LIN {X 0,Y 419.556,Z 514.347,A -85,B 0,C 180,E1 -10185.297,E2 -10185.297} C_VEL
LIN {X 0,Y 420.532,Z 504.922,A -85,B 0,C 180,E1 -10186.755,E2 -10186.755} C_VEL
LIN {X 0,Y 421.766,Z 492.891,A -85,B 0,C 180,E1 -10188.309,E2 -10188.309} C_VEL
LIN {X 0,Y 423.026,Z 480.248,A -85,B 0,C 180,E1 -10189.659,E2 -10189.659} C_VEL
LIN {X 0,Y 424.183,Z 467.994,A -85,B 0,C 180,E1 -10190.741,E2 -10190.741} C_VEL
LIN {X 0,Y 425.391,Z 454.765,A -85,B 0,C 180,E1 -10191.694,E2 -10191.694} C_VEL
LIN {X 0,Y 426.558,Z 439.892,A -85,B 0,C 180,E1 -10192.546,E2 -10192.546} C_VEL
LIN {X 0,Y 427.411,Z 424.917,A -85,B 0,C 180,E1 -10193.196,E2 -10193.196} C_VEL
LIN {X 0,Y 428.173,Z 409.767,A -85,B 0,C 180,E1 -10193.647,E2 -10193.647} C_VEL
LIN {X 0,Y 428.857,Z 376.254,A -85,B 0,C 180,E1 -10194.249,E2 -10194.249} C_VEL
LIN {X 0,Y 430.577,Z 275.254,A -85,B 0,C 180,E1 -10195.966,E2 -10195.966} C_VEL
LIN {X 0,Y 425.192,Z 246.932,A -85,B 0,C 180,E1 -10196.839,E2 -10196.839} C_VEL
LIN {X 0,Y 424.129,Z 241.646,A -85,B 0,C 180,E1 -10197.03,E2 -10197.03} C_VEL
LIN {X 0,Y 424.477,Z 235.443,A -85,B 0,C 180,E1 -10198.074,E2 -10198.074} C_VEL
LIN {X 0,Y 421.44,Z 222.358,A -85,B 0,C 180,E1 -10200.571,E2 -10200.571} C_VEL
LIN {X 0,Y 418.245,Z 209.999,A -85,B 0,C 180,E1 -10203.07,E2 -10203.07} C_VEL
LIN {X 0,Y 418.245,Z 210.011,A -85,B 0,C 180,E1 -10206.238,E2 -10206.238} C_VEL
LIN {X 0,Y 418.26,Z 210.01,A -85,B 0,C 180,E1 -10209.68,E2 -10209.68} C_VEL
LIN {X 0,Y 418.241,Z 210.012,A -85,B 0,C 180,E1 -10212.323,E2 -10212.323} C_VEL
LIN {X 0,Y 418.23,Z 210.009,A -85,B 0,C 180,E1 -10215.108,E2 -10215.108} C_VEL
LIN {X 0,Y 418.251,Z 210.009,A -85,B 0,C 180,E1 -10217.768,E2 -10217.768} C_VEL
LIN {X 0,Y 418.261,Z 210.005,A -85,B 0,C 180,E1 -10220.616,E2 -10220.616} C_VEL
LIN {X 0,Y 418.24,Z 210.008,A -85,B 0,C 180,E1 -10223.976,E2 -10223.976} C_VEL
LIN {X 0,Y 418.253,Z 210.004,A -85,B 0,C 180,E1 -10227.155,E2 -10227.155} C_VEL
LIN {X 0,Y 418.267,Z 210.003,A -85,B 0,C 180,E1 -10230.838,E2 -10230.838} C_VEL
LIN {X 0,Y 418.263,Z 210.01,A -85,B 0,C 180,E1 -10234.096,E2 -10234.096} C_VEL
LIN {X 0,Y 418.224,Z 210.004,A -85,B 0,C 180,E1 -10237.263,E2 -10237.263} C_VEL
LIN {X 0,Y 418.275,Z 210.003,A -85,B 0,C 180,E1 -10240.364,E2 -10240.364} C_VEL
LIN {X 0,Y 418.308,Z 210.002,A -85,B 0,C 180,E1 -10243.404,E2 -10243.404} C_VEL
LIN {X 0,Y 418.338,Z 209.997,A -85,B 0,C 180,E1 -10246.999,E2 -10246.999} C_VEL
LIN {X 0,Y 418.334,Z 209.997,A -85,B 0,C 180,E1 -10250.329,E2 -10250.329} C_VEL
LIN {X 0,Y 418.484,Z 209.981,A -85,B 0,C 180,E1 -10253.249,E2 -10253.249} C_VEL
LIN {X 0,Y 418.333,Z 210,A -85,B 0,C 180,E1 -10255.182,E2 -10255.182} C_VEL
LIN {X 0,Y 418.536,Z 209.973,A -85,B 0,C 180,E1 -10258.076,E2 -10258.076} C_VEL
LIN {X 0,Y 418.665,Z 209.953,A -85,B 0,C 180,E1 -10260,E2 -10260} C_VEL
LIN {X 0,Y 418.503,Z 209.979,A -85,B 0,C 180,E1 -10262.888,E2 -10262.888} C_VEL
LIN {X 0,Y 418.486,Z 209.98,A -85,B 0,C 180,E1 -10266.751,E2 -10266.751} C_VEL
LIN {X 0,Y 418.334,Z 210,A -85,B 0,C 180,E1 -10269.672,E2 -10269.672} C_VEL
LIN {X 0,Y 418.339,Z 209.996,A -85,B 0,C 180,E1 -10273.001,E2 -10273.001} C_VEL
LIN {X 0,Y 418.305,Z 210.001,A -85,B 0,C 180,E1 -10276.736,E2 -10276.736} C_VEL
LIN {X 0,Y 418.263,Z 210.005,A -85,B 0,C 180,E1 -10279.791,E2 -10279.791} C_VEL
LIN {X 0,Y 418.225,Z 210.014,A -85,B 0,C 180,E1 -10282.737,E2 -10282.737} C_VEL
LIN {X 0,Y 418.263,Z 209.987,A -85,B 0,C 180,E1 -10285.905,E2 -10285.905} C_VEL
LIN {X 0,Y 418.269,Z 210.011,A -85,B 0,C 180,E1 -10289.162,E2 -10289.162} C_VEL
LIN {X 0,Y 418.252,Z 210.013,A -85,B 0,C 180,E1 -10292.845,E2 -10292.845} C_VEL
LIN {X 0,Y 418.243,Z 210.009,A -85,B 0,C 180,E1 -10296.239,E2 -10296.239} C_VEL
LIN {X 0,Y 418.244,Z 210.006,A -85,B 0,C 180,E1 -10299.683,E2 -10299.683} C_VEL
LIN {X 0,Y 418.227,Z 210.009,A -85,B 0,C 180,E1 -10302.322,E2 -10302.322} C_VEL
LIN {X 0,Y 418.238,Z 210.013,A -85,B 0,C 180,E1 -10305.11,E2 -10305.11} C_VEL
LIN {X 0,Y 418.239,Z 210.011,A -85,B 0,C 180,E1 -10307.768,E2 -10307.768} C_VEL
LIN {X 0,Y 418.255,Z 210.007,A -85,B 0,C 180,E1 -10310.619,E2 -10310.619} C_VEL
LIN {X 0,Y 418.24,Z 210.008,A -85,B 0,C 180,E1 -10313.977,E2 -10313.977} C_VEL
LIN {X 0,Y 418.256,Z 210.009,A -85,B 0,C 180,E1 -10317.157,E2 -10317.157} C_VEL
LIN {X 0,Y 418.269,Z 210.134,A -85,B 0,C 180,E1 -10320.425,E2 -10320.425} C_VEL
LIN {X 0,Y 421.107,Z 221.313,A -85,B 0,C 180,E1 -10322.844,E2 -10322.844} C_VEL
LIN {X 0,Y 429.206,Z 240.547,A -85,B 0,C 180,E1 -10323.755,E2 -10323.755} C_VEL
LIN {X 0,Y 430.885,Z 248.586,A -85,B 0,C 180,E1 -10324.013,E2 -10324.013} C_VEL
LIN {X 0,Y 429.161,Z 353.4,A -85,B 0,C 180,E1 -10325.801,E2 -10325.801} C_VEL
LIN {X 0,Y 428.505,Z 387.1,A -85,B 0,C 180,E1 -10326.404,E2 -10326.404} C_VEL
LIN {X 0,Y 427.927,Z 402.384,A -85,B 0,C 180,E1 -10326.867,E2 -10326.867} C_VEL
LIN {X 0,Y 427.22,Z 415.712,A -85,B 0,C 180,E1 -10327.435,E2 -10327.435} C_VEL
LIN {X 0,Y 426.193,Z 429.869,A -85,B 0,C 180,E1 -10328.221,E2 -10328.221} C_VEL
LIN {X 0,Y 425.1,Z 443.449,A -85,B 0,C 180,E1 -10329.179,E2 -10329.179} C_VEL
LIN {X 0,Y 423.774,Z 457.224,A -85,B 0,C 180,E1 -10330.377,E2 -10330.377} C_VEL
LIN {X 0,Y 422.655,Z 468.581,A -85,B 0,C 180,E1 -10331.583,E2 -10331.583} C_VEL
LIN {X 0,Y 421.421,Z 480.043,A -85,B 0,C 180,E1 -10333.032,E2 -10333.032} C_VEL
LIN {X 0,Y 421.245,Z 481.801,A -85,B 0,C 180,E1 -10333.273,E2 -10333.273} C_VEL
LIN {X 0,Y 420.192,Z 485.905,A -85,B 0,C 180,E1 -10333.835,E2 -10333.835} C_VEL
LIN {X 0,Y 416.726,Z 492.332,A -85,B 0,C 180,E1 -10334.755,E2 -10334.755} C_VEL
LIN {X 0,Y 413.246,Z 498.267,A -85,B 0,C 180,E1 -10335.744,E2 -10335.744} C_VEL
LIN {X 0,Y 412.186,Z 501.6,A -85,B 0,C 180,E1 -10336.407,E2 -10336.407} C_VEL
LIN {X 0,Y 411.566,Z 509.194,A -85,B 0,C 180,E1 -10338.176,E2 -10338.176} C_VEL
LIN {X 0,Y 410.838,Z 516.135,A -85,B 0,C 180,E1 -10340.15,E2 -10340.15} C_VEL
LIN {X 0,Y 410.44,Z 521.585,A -85,B 0,C 180,E1 -10342.127,E2 -10342.127} C_VEL
LIN {X 0,Y 410.201,Z 525.699,A -85,B 0,C 180,E1 -10344.1,E2 -10344.1} C_VEL
LIN {X 0,Y 409.982,Z 528.593,A -85,B 0,C 180,E1 -10346.068,E2 -10346.068} C_VEL
LIN {X 0,Y 410.007,Z 530.331,A -85,B 0,C 180,E1 -10348.035,E2 -10348.035} C_VEL
LIN {X 0,Y 409.925,Z 530.941,A -85,B 0,C 180,E1 -10350,E2 -10350} C_VEL
LIN {X 0,Y 410.008,Z 530.379,A -85,B 0,C 180,E1 -10351.965,E2 -10351.965} C_VEL
LIN {X 0,Y 409.981,Z 528.706,A -85,B 0,C 180,E1 -10353.932,E2 -10353.932} C_VEL
LIN {X 0,Y 410.185,Z 525.873,A -85,B 0,C 180,E1 -10355.9,E2 -10355.9} C_VEL
LIN {X 0,Y 410.411,Z 521.819,A -85,B 0,C 180,E1 -10357.874,E2 -10357.874} C_VEL
LIN {X 0,Y 410.824,Z 516.442,A -85,B 0,C 180,E1 -10359.85,E2 -10359.85} C_VEL
LIN {X 0,Y 411.55,Z 509.585,A -85,B 0,C 180,E1 -10361.825,E2 -10361.825} C_VEL
LIN {X 0,Y 412.292,Z 501.03,A -85,B 0,C 180,E1 -10363.806,E2 -10363.806} C_VEL
LIN {X 0,Y 413.317,Z 491.928,A -85,B 0,C 180,E1 -10365.534,E2 -10365.534} C_VEL
LIN {X 0,Y 414.339,Z 482.65,A -85,B 0,C 180,E1 -10367.013,E2 -10367.013} C_VEL
LIN {X 0,Y 415.663,Z 470.729,A -85,B 0,C 180,E1 -10368.6,E2 -10368.6} C_VEL
LIN {X 0,Y 417.002,Z 458.382,A -85,B 0,C 180,E1 -10369.955,E2 -10369.955} C_VEL
LIN {X 0,Y 418.359,Z 444.849,A -85,B 0,C 180,E1 -10371.172,E2 -10371.172} C_VEL
LIN {X 0,Y 419.529,Z 431.537,A -85,B 0,C 180,E1 -10372.143,E2 -10372.143} C_VEL
LIN {X 0,Y 420.595,Z 416.874,A -85,B 0,C 180,E1 -10372.988,E2 -10372.988} C_VEL
LIN {X 0,Y 421.415,Z 402.214,A -85,B 0,C 180,E1 -10373.626,E2 -10373.626} C_VEL
LIN {X 0,Y 422.043,Z 387.314,A -85,B 0,C 180,E1 -10374.077,E2 -10374.077} C_VEL
LIN {X 0,Y 422.876,Z 348.258,A -85,B 0,C 180,E1 -10374.779,E2 -10374.779} C_VEL
LIN {X 0,Y 424.496,Z 248.846,A -85,B 0,C 180,E1 -10376.506,E2 -10376.506} C_VEL
LIN {X 0,Y 422.718,Z 241.83,A -85,B 0,C 180,E1 -10376.758,E2 -10376.758} C_VEL
LIN {X 0,Y 414.382,Z 222.693,A -85,B 0,C 180,E1 -10377.712,E2 -10377.712} C_VEL
LIN {X 0,Y 413.816,Z 221.203,A -85,B 0,C 180,E1 -10377.806,E2 -10377.806} C_VEL
LIN {X 0,Y 411.215,Z 210.89,A -85,B 0,C 180,E1 -10380.134,E2 -10380.134} C_VEL
LIN {X 0,Y 411.205,Z 210.895,A -85,B 0,C 180,E1 -10383.155,E2 -10383.155} C_VEL
LIN {X 0,Y 411.193,Z 210.888,A -85,B 0,C 180,E1 -10386.552,E2 -10386.552} C_VEL
LIN {X 0,Y 411.211,Z 210.883,A -85,B 0,C 180,E1 -10389.727,E2 -10389.727} C_VEL
LIN {X 0,Y 411.174,Z 210.894,A -85,B 0,C 180,E1 -10393.132,E2 -10393.132} C_VEL
LIN {X 0,Y 411.164,Z 210.891,A -85,B 0,C 180,E1 -10395.88,E2 -10395.88} C_VEL
LIN {X 0,Y 411.195,Z 210.883,A -85,B 0,C 180,E1 -10398.765,E2 -10398.765} C_VEL
LIN {X 0,Y 411.198,Z 210.876,A -85,B 0,C 180,E1 -10402.027,E2 -10402.027} C_VEL
LIN {X 0,Y 411.2,Z 210.888,A -85,B 0,C 180,E1 -10405.666,E2 -10405.666} C_VEL
LIN {X 0,Y 411.191,Z 210.874,A -85,B 0,C 180,E1 -10409.152,E2 -10409.152} C_VEL
LIN {X 0,Y 411.253,Z 210.882,A -85,B 0,C 180,E1 -10412.522,E2 -10412.522} C_VEL
LIN {X 0,Y 411.219,Z 210.884,A -85,B 0,C 180,E1 -10415.784,E2 -10415.784} C_VEL
LIN {X 0,Y 411.188,Z 210.892,A -85,B 0,C 180,E1 -10418.965,E2 -10418.965} C_VEL
LIN {X 0,Y 411.245,Z 210.877,A -85,B 0,C 180,E1 -10422.084,E2 -10422.084} C_VEL
LIN {X 0,Y 411.252,Z 210.877,A -85,B 0,C 180,E1 -10425.147,E2 -10425.147} C_VEL
LIN {X 0,Y 411.277,Z 210.878,A -85,B 0,C 180,E1 -10428.167,E2 -10428.167} C_VEL
LIN {X 0,Y 411.432,Z 210.858,A -85,B 0,C 180,E1 -10432.189,E2 -10432.189} C_VEL
LIN {X 0,Y 411.466,Z 210.852,A -85,B 0,C 180,E1 -10434.118,E2 -10434.118} C_VEL
LIN {X 0,Y 411.505,Z 210.849,A -85,B 0,C 180,E1 -10438.042,E2 -10438.042} C_VEL
LIN {X 0,Y 411.635,Z 210.827,A -85,B 0,C 180,E1 -10440,E2 -10440} C_VEL
LIN {X 0,Y 411.458,Z 210.853,A -85,B 0,C 180,E1 -10442.937,E2 -10442.937} C_VEL
LIN {X 0,Y 411.447,Z 210.857,A -85,B 0,C 180,E1 -10446.867,E2 -10446.867} C_VEL
LIN {X 0,Y 411.285,Z 210.875,A -85,B 0,C 180,E1 -10449.839,E2 -10449.839} C_VEL
LIN {X 0,Y 411.297,Z 210.872,A -85,B 0,C 180,E1 -10453.104,E2 -10453.104} C_VEL
LIN {X 0,Y 411.255,Z 210.883,A -85,B 0,C 180,E1 -10455.868,E2 -10455.868} C_VEL
LIN {X 0,Y 411.217,Z 210.888,A -85,B 0,C 180,E1 -10458.949,E2 -10458.949} C_VEL
LIN {X 0,Y 411.196,Z 210.892,A -85,B 0,C 180,E1 -10462.643,E2 -10462.643} C_VEL
LIN {X 0,Y 411.229,Z 210.88,A -85,B 0,C 180,E1 -10465.293,E2 -10465.293} C_VEL
LIN {X 0,Y 411.217,Z 210.889,A -85,B 0,C 180,E1 -10468.59,E2 -10468.59} C_VEL
LIN {X 0,Y 411.164,Z 210.894,A -85,B 0,C 180,E1 -10471.997,E2 -10471.997} C_VEL
LIN {X 0,Y 411.192,Z 210.888,A -85,B 0,C 180,E1 -10475.529,E2 -10475.529} C_VEL
LIN {X 0,Y 411.212,Z 210.881,A -85,B 0,C 180,E1 -10479.225,E2 -10479.225} C_VEL
LIN {X 0,Y 411.176,Z 210.892,A -85,B 0,C 180,E1 -10482.696,E2 -10482.696} C_VEL
LIN {X 0,Y 411.163,Z 210.895,A -85,B 0,C 180,E1 -10485.882,E2 -10485.882} C_VEL
LIN {X 0,Y 411.196,Z 210.888,A -85,B 0,C 180,E1 -10488.766,E2 -10488.766} C_VEL
LIN {X 0,Y 411.2,Z 210.882,A -85,B 0,C 180,E1 -10492.028,E2 -10492.028} C_VEL
LIN {X 0,Y 411.203,Z 210.89,A -85,B 0,C 180,E1 -10495.667,E2 -10495.667} C_VEL
LIN {X 0,Y 411.209,Z 210.944,A -85,B 0,C 180,E1 -10496.516,E2 -10496.516} C_VEL
LIN {X 0,Y 415.204,Z 226.483,A -85,B 0,C 180,E1 -10499.684,E2 -10499.684} C_VEL
LIN {X 0,Y 417.712,Z 237.94,A -85,B 0,C 180,E1 -10501.895,E2 -10501.895} C_VEL
LIN {X 0,Y 417.473,Z 241.807,A -85,B 0,C 180,E1 -10502.522,E2 -10502.522} C_VEL
LIN {X 0,Y 423.749,Z 273.294,A -85,B 0,C 180,E1 -10503.543,E2 -10503.543} C_VEL
LIN {X 0,Y 424.228,Z 277.071,A -85,B 0,C 180,E1 -10503.645,E2 -10503.645} C_VEL
LIN {X 0,Y 421.757,Z 407.384,A -85,B 0,C 180,E1 -10505.905,E2 -10505.905} C_VEL
LIN {X 0,Y 421.078,Z 422.903,A -85,B 0,C 180,E1 -10506.354,E2 -10506.354} C_VEL
LIN {X 0,Y 420.16,Z 437.166,A -85,B 0,C 180,E1 -10506.95,E2 -10506.95} C_VEL
LIN {X 0,Y 419.122,Z 450.867,A -85,B 0,C 180,E1 -10507.705,E2 -10507.705} C_VEL
LIN {X 0,Y 417.804,Z 464.768,A -85,B 0,C 180,E1 -10508.669,E2 -10508.669} C_VEL
LIN {X 0,Y 416.602,Z 477.512,A -85,B 0,C 180,E1 -10509.768,E2 -10509.768} C_VEL
LIN {X 0,Y 415.151,Z 490.399,A -85,B 0,C 180,E1 -10511.11,E2 -10511.11} C_VEL
LIN {X 0,Y 414.054,Z 501.198,A -85,B 0,C 180,E1 -10512.466,E2 -10512.466} C_VEL
LIN {X 0,Y 412.908,Z 511.188,A -85,B 0,C 180,E1 -10513.944,E2 -10513.944} C_VEL
LIN {X 0,Y 411.914,Z 520.968,A -85,B 0,C 180,E1 -10515.677,E2 -10515.677} C_VEL
LIN {X 0,Y 411.211,Z 529.133,A -85,B 0,C 180,E1 -10517.414,E2 -10517.414} C_VEL
LIN {X 0,Y 410.667,Z 535.884,A -85,B 0,C 180,E1 -10519.15,E2 -10519.15} C_VEL
LIN {X 0,Y 410.235,Z 542.121,A -85,B 0,C 180,E1 -10521.131,E2 -10521.131} C_VEL
LIN {X 0,Y 410.056,Z 546.949,A -85,B 0,C 180,E1 -10523.11,E2 -10523.11} C_VEL
LIN {X 0,Y 409.935,Z 550.485,A -85,B 0,C 180,E1 -10525.083,E2 -10525.083} C_VEL
LIN {X 0,Y 409.903,Z 552.813,A -85,B 0,C 180,E1 -10527.052,E2 -10527.052} C_VEL
LIN {X 0,Y 409.933,Z 553.984,A -85,B 0,C 180,E1 -10529.018,E2 -10529.018} C_VEL
LIN {X 0,Y 409.933,Z 553.983,A -85,B 0,C 180,E1 -10530.982,E2 -10530.982} C_VEL
LIN {X 0,Y 409.903,Z 552.804,A -85,B 0,C 180,E1 -10532.948,E2 -10532.948} C_VEL
LIN {X 0,Y 409.939,Z 550.474,A -85,B 0,C 180,E1 -10534.917,E2 -10534.917} C_VEL
LIN {X 0,Y 410.06,Z 546.939,A -85,B 0,C 180,E1 -10536.89,E2 -10536.89} C_VEL
LIN {X 0,Y 410.235,Z 542.11,A -85,B 0,C 180,E1 -10538.869,E2 -10538.869} C_VEL
LIN {X 0,Y 410.667,Z 535.86,A -85,B 0,C 180,E1 -10540.85,E2 -10540.85} C_VEL
LIN {X 0,Y 411.177,Z 529.103,A -85,B 0,C 180,E1 -10542.587,E2 -10542.587} C_VEL
LIN {X 0,Y 411.912,Z 520.937,A -85,B 0,C 180,E1 -10544.323,E2 -10544.323} C_VEL
LIN {X 0,Y 412.912,Z 511.152,A -85,B 0,C 180,E1 -10546.056,E2 -10546.056} C_VEL
LIN {X 0,Y 414.048,Z 501.152,A -85,B 0,C 180,E1 -10547.534,E2 -10547.534} C_VEL
LIN {X 0,Y 415.294,Z 489.277,A -85,B 0,C 180,E1 -10549.012,E2 -10549.012} C_VEL
LIN {X 0,Y 416.592,Z 477.449,A -85,B 0,C 180,E1 -10550.233,E2 -10550.233} C_VEL
LIN {X 0,Y 417.846,Z 464.677,A -85,B 0,C 180,E1 -10551.329,E2 -10551.329} C_VEL
LIN {X 0,Y 419.092,Z 450.747,A -85,B 0,C 180,E1 -10552.297,E2 -10552.297} C_VEL
LIN {X 0,Y 420.238,Z 435.912,A -85,B 0,C 180,E1 -10553.102,E2 -10553.102} C_VEL
LIN {X 0,Y 421.135,Z 420.871,A -85,B 0,C 180,E1 -10553.708,E2 -10553.708} C_VEL
LIN {X 0,Y 421.828,Z 405.525,A -85,B 0,C 180,E1 -10554.123,E2 -10554.123} C_VEL
LIN {X 0,Y 424.192,Z 276.094,A -85,B 0,C 180,E1 -10556.367,E2 -10556.367} C_VEL
LIN {X 0,Y 418.811,Z 248.109,A -85,B 0,C 180,E1 -10557.255,E2 -10557.255} C_VEL
LIN {X 0,Y 417.458,Z 241.434,A -85,B 0,C 180,E1 -10557.499,E2 -10557.499} C_VEL
LIN {X 0,Y 417.705,Z 237.876,A -85,B 0,C 180,E1 -10558.106,E2 -10558.106} C_VEL
LIN {X 0,Y 415.22,Z 226.384,A -85,B 0,C 180,E1 -10560.32,E2 -10560.32} C_VEL
LIN {X 0,Y 411.212,Z 210.874,A -85,B 0,C 180,E1 -10563.52,E2 -10563.52} C_VEL
LIN {X 0,Y 411.19,Z 210.89,A -85,B 0,C 180,E1 -10566.741,E2 -10566.741} C_VEL
LIN {X 0,Y 411.223,Z 210.886,A -85,B 0,C 180,E1 -10569.729,E2 -10569.729} C_VEL
LIN {X 0,Y 411.173,Z 210.889,A -85,B 0,C 180,E1 -10573.132,E2 -10573.132} C_VEL
LIN {X 0,Y 411.163,Z 210.894,A -85,B 0,C 180,E1 -10575.88,E2 -10575.88} C_VEL
LIN {X 0,Y 411.194,Z 210.885,A -85,B 0,C 180,E1 -10578.765,E2 -10578.765} C_VEL
LIN {X 0,Y 411.198,Z 210.886,A -85,B 0,C 180,E1 -10582.027,E2 -10582.027} C_VEL
LIN {X 0,Y 411.2,Z 210.887,A -85,B 0,C 180,E1 -10585.666,E2 -10585.666} C_VEL
LIN {X 0,Y 411.193,Z 210.886,A -85,B 0,C 180,E1 -10589.153,E2 -10589.153} C_VEL
LIN {X 0,Y 411.253,Z 210.877,A -85,B 0,C 180,E1 -10592.522,E2 -10592.522} C_VEL
LIN {X 0,Y 411.213,Z 210.886,A -85,B 0,C 180,E1 -10595.784,E2 -10595.784} C_VEL
LIN {X 0,Y 411.188,Z 210.872,A -85,B 0,C 180,E1 -10598.966,E2 -10598.966} C_VEL
LIN {X 0,Y 411.244,Z 210.882,A -85,B 0,C 180,E1 -10602.085,E2 -10602.085} C_VEL
LIN {X 0,Y 411.251,Z 210.881,A -85,B 0,C 180,E1 -10605.147,E2 -10605.147} C_VEL
LIN {X 0,Y 411.276,Z 210.876,A -85,B 0,C 180,E1 -10608.167,E2 -10608.167} C_VEL
LIN {X 0,Y 411.432,Z 210.856,A -85,B 0,C 180,E1 -10612.189,E2 -10612.189} C_VEL
LIN {X 0,Y 411.466,Z 210.853,A -85,B 0,C 180,E1 -10614.118,E2 -10614.118} C_VEL
LIN {X 0,Y 411.505,Z 210.849,A -85,B 0,C 180,E1 -10618.043,E2 -10618.043} C_VEL
LIN {X 0,Y 411.635,Z 210.828,A -85,B 0,C 180,E1 -10620,E2 -10620} C_VEL
LIN {X 0,Y 411.458,Z 210.857,A -85,B 0,C 180,E1 -10622.937,E2 -10622.937} C_VEL
LIN {X 0,Y 411.453,Z 210.857,A -85,B 0,C 180,E1 -10626.867,E2 -10626.867} C_VEL
LIN {X 0,Y 411.286,Z 210.877,A -85,B 0,C 180,E1 -10629.839,E2 -10629.839} C_VEL
LIN {X 0,Y 411.298,Z 210.873,A -85,B 0,C 180,E1 -10633.105,E2 -10633.105} C_VEL
LIN {X 0,Y 411.255,Z 210.879,A -85,B 0,C 180,E1 -10636.869,E2 -10636.869} C_VEL
LIN {X 0,Y 411.223,Z 210.881,A -85,B 0,C 180,E1 -10639.987,E2 -10639.987} C_VEL
LIN {X 0,Y 411.189,Z 210.891,A -85,B 0,C 180,E1 -10643.148,E2 -10643.148} C_VEL
LIN {X 0,Y 411.231,Z 210.863,A -85,B 0,C 180,E1 -10646.381,E2 -10646.381} C_VEL
LIN {X 0,Y 411.205,Z 210.886,A -85,B 0,C 180,E1 -10649.712,E2 -10649.712} C_VEL
LIN {X 0,Y 411.201,Z 210.887,A -85,B 0,C 180,E1 -10653.156,E2 -10653.156} C_VEL
LIN {X 0,Y 411.19,Z 210.889,A -85,B 0,C 180,E1 -10656.554,E2 -10656.554} C_VEL
LIN {X 0,Y 411.208,Z 210.882,A -85,B 0,C 180,E1 -10659.729,E2 -10659.729} C_VEL
LIN {X 0,Y 411.173,Z 210.891,A -85,B 0,C 180,E1 -10663.134,E2 -10663.134} C_VEL
LIN {X 0,Y 411.17,Z 210.89,A -85,B 0,C 180,E1 -10665.881,E2 -10665.881} C_VEL
LIN {X 0,Y 411.163,Z 210.896,A -85,B 0,C 180,E1 -10668.772,E2 -10668.772} C_VEL
LIN {X 0,Y 411.204,Z 210.886,A -85,B 0,C 180,E1 -10671.832,E2 -10671.832} C_VEL
LIN {X 0,Y 411.208,Z 210.891,A -85,B 0,C 180,E1 -10675.122,E2 -10675.122} C_VEL
LIN {X 0,Y 411.164,Z 210.896,A -85,B 0,C 180,E1 -10678.003,E2 -10678.003} C_VEL
LIN {X 0,Y 411.239,Z 211.022,A -85,B 0,C 180,E1 -10680.009,E2 -10680.009} C_VEL
LIN {X 0,Y 413.982,Z 221.604,A -85,B 0,C 180,E1 -10682.338,E2 -10682.338} C_VEL
LIN {X 0,Y 423.128,Z 243.066,A -85,B 0,C 180,E1 -10683.392,E2 -10683.392} C_VEL
LIN {X 0,Y 424.523,Z 249.367,A -85,B 0,C 180,E1 -10683.604,E2 -10683.604} C_VEL
LIN {X 0,Y 422.698,Z 353.627,A -85,B 0,C 180,E1 -10685.407,E2 -10685.407} C_VEL
LIN {X 0,Y 422.011,Z 387.317,A -85,B 0,C 180,E1 -10686.018,E2 -10686.018} C_VEL
LIN {X 0,Y 421.407,Z 402.714,A -85,B 0,C 180,E1 -10686.492,E2 -10686.492} C_VEL
LIN {X 0,Y 420.653,Z 416.329,A -85,B 0,C 180,E1 -10687.083,E2 -10687.083} C_VEL
LIN {X 0,Y 419.607,Z 430.077,A -85,B 0,C 180,E1 -10687.862,E2 -10687.862} C_VEL
LIN {X 0,Y 418.479,Z 443.656,A -85,B 0,C 180,E1 -10688.834,E2 -10688.834} C_VEL
LIN {X 0,Y 417.067,Z 457.431,A -85,B 0,C 180,E1 -10690.048,E2 -10690.048} C_VEL
LIN {X 0,Y 415.783,Z 469.85,A -85,B 0,C 180,E1 -10691.395,E2 -10691.395} C_VEL
LIN {X 0,Y 414.618,Z 480.247,A -85,B 0,C 180,E1 -10692.745,E2 -10692.745} C_VEL
LIN {X 0,Y 413.534,Z 489.888,A -85,B 0,C 180,E1 -10694.222,E2 -10694.222} C_VEL
LIN {X 0,Y 412.463,Z 499.336,A -85,B 0,C 180,E1 -10695.948,E2 -10695.948} C_VEL
LIN {X 0,Y 412.186,Z 501.6,A -85,B 0,C 180,E1 -10696.407,E2 -10696.407} C_VEL
LIN {X 0,Y 411.167,Z 504.821,A -85,B 0,C 180,E1 -10697.086,E2 -10697.086} C_VEL
LIN {X 0,Y 407.865,Z 509.804,A -85,B 0,C 180,E1 -10698.194,E2 -10698.194} C_VEL
LIN {X 0,Y 404.646,Z 514.3,A -85,B 0,C 180,E1 -10699.354,E2 -10699.354} C_VEL
LIN {X 0,Y 403.77,Z 516.725,A -85,B 0,C 180,E1 -10700.108,E2 -10700.108} C_VEL
LIN {X 0,Y 403.388,Z 521.787,A -85,B 0,C 180,E1 -10701.988,E2 -10701.988} C_VEL
LIN {X 0,Y 403.122,Z 525.901,A -85,B 0,C 180,E1 -10703.996,E2 -10703.996} C_VEL
LIN {X 0,Y 402.902,Z 528.794,A -85,B 0,C 180,E1 -10705.999,E2 -10705.999} C_VEL
LIN {X 0,Y 402.921,Z 530.531,A -85,B 0,C 180,E1 -10708.001,E2 -10708.001} C_VEL
LIN {X 0,Y 402.85,Z 531.141,A -85,B 0,C 180,E1 -10710,E2 -10710} C_VEL
LIN {X 0,Y 402.921,Z 530.579,A -85,B 0,C 180,E1 -10711.999,E2 -10711.999} C_VEL
LIN {X 0,Y 402.901,Z 528.906,A -85,B 0,C 180,E1 -10714.001,E2 -10714.001} C_VEL
LIN {X 0,Y 403.109,Z 526.073,A -85,B 0,C 180,E1 -10716.004,E2 -10716.004} C_VEL
LIN {X 0,Y 403.366,Z 522.019,A -85,B 0,C 180,E1 -10718.012,E2 -10718.012} C_VEL
LIN {X 0,Y 403.794,Z 516.643,A -85,B 0,C 180,E1 -10720.023,E2 -10720.023} C_VEL
LIN {X 0,Y 404.586,Z 509.785,A -85,B 0,C 180,E1 -10722.031,E2 -10722.031} C_VEL
LIN {X 0,Y 405.386,Z 501.229,A -85,B 0,C 180,E1 -10724.046,E2 -10724.046} C_VEL
LIN {X 0,Y 406.436,Z 492.127,A -85,B 0,C 180,E1 -10725.803,E2 -10725.803} C_VEL
LIN {X 0,Y 407.518,Z 482.849,A -85,B 0,C 180,E1 -10727.307,E2 -10727.307} C_VEL
LIN {X 0,Y 408.843,Z 471.501,A -85,B 0,C 180,E1 -10728.846,E2 -10728.846} C_VEL
LIN {X 0,Y 410.335,Z 458.579,A -85,B 0,C 180,E1 -10730.293,E2 -10730.293} C_VEL
LIN {X 0,Y 411.716,Z 445.045,A -85,B 0,C 180,E1 -10731.53,E2 -10731.53} C_VEL
LIN {X 0,Y 412.968,Z 431.731,A -85,B 0,C 180,E1 -10732.514,E2 -10732.514} C_VEL
LIN {X 0,Y 414.105,Z 416.59,A -85,B 0,C 180,E1 -10733.396,E2 -10733.396} C_VEL
LIN {X 0,Y 414.969,Z 401.595,A -85,B 0,C 180,E1 -10734.049,E2 -10734.049} C_VEL
LIN {X 0,Y 415.631,Z 386.311,A -85,B 0,C 180,E1 -10734.506,E2 -10734.506} C_VEL
LIN {X 0,Y 417.65,Z 282.682,A -85,B 0,C 180,E1 -10736.341,E2 -10736.341} C_VEL
LIN {X 0,Y 418.218,Z 250.264,A -85,B 0,C 180,E1 -10736.913,E2 -10736.913} C_VEL
LIN {X 0,Y 416.588,Z 244.136,A -85,B 0,C 180,E1 -10737.144,E2 -10737.144} C_VEL
LIN {X 0,Y 407.787,Z 224.161,A -85,B 0,C 180,E1 -10738.175,E2 -10738.175} C_VEL
LIN {X 0,Y 406.59,Z 221.401,A -85,B 0,C 180,E1 -10738.349,E2 -10738.349} C_VEL
LIN {X 0,Y 404.156,Z 211.768,A -85,B 0,C 180,E1 -10740.572,E2 -10740.572} C_VEL
LIN {X 0,Y 404.143,Z 211.768,A -85,B 0,C 180,E1 -10743.812,E2 -10743.812} C_VEL
LIN {X 0,Y 404.137,Z 211.767,A -85,B 0,C 180,E1 -10746.875,E2 -10746.875} C_VEL
LIN {X 0,Y 404.144,Z 211.763,A -85,B 0,C 180,E1 -10750.079,E2 -10750.079} C_VEL
LIN {X 0,Y 404.153,Z 211.768,A -85,B 0,C 180,E1 -10753.084,E2 -10753.084} C_VEL
LIN {X 0,Y 404.144,Z 211.766,A -85,B 0,C 180,E1 -10755.925,E2 -10755.925} C_VEL
LIN {X 0,Y 404.147,Z 211.76,A -85,B 0,C 180,E1 -10758.638,E2 -10758.638} C_VEL
LIN {X 0,Y 404.156,Z 211.756,A -85,B 0,C 180,E1 -10761.49,E2 -10761.49} C_VEL
LIN {X 0,Y 404.18,Z 211.763,A -85,B 0,C 180,E1 -10764.983,E2 -10764.983} C_VEL
LIN {X 0,Y 404.139,Z 211.749,A -85,B 0,C 180,E1 -10768.553,E2 -10768.553} C_VEL
LIN {X 0,Y 404.191,Z 211.76,A -85,B 0,C 180,E1 -10772,E2 -10772} C_VEL
LIN {X 0,Y 404.17,Z 211.766,A -85,B 0,C 180,E1 -10775.334,E2 -10775.334} C_VEL
LIN {X 0,Y 404.131,Z 211.766,A -85,B 0,C 180,E1 -10778.58,E2 -10778.58} C_VEL
LIN {X 0,Y 404.202,Z 211.754,A -85,B 0,C 180,E1 -10781.761,E2 -10781.761} C_VEL
LIN {X 0,Y 404.198,Z 211.758,A -85,B 0,C 180,E1 -10784.882,E2 -10784.882} C_VEL
LIN {X 0,Y 404.249,Z 211.753,A -85,B 0,C 180,E1 -10787.958,E2 -10787.958} C_VEL
LIN {X 0,Y 404.397,Z 211.734,A -85,B 0,C 180,E1 -10792.128,E2 -10792.128} C_VEL
LIN {X 0,Y 404.414,Z 211.73,A -85,B 0,C 180,E1 -10794.015,E2 -10794.015} C_VEL
LIN {X 0,Y 404.474,Z 211.725,A -85,B 0,C 180,E1 -10798.008,E2 -10798.008} C_VEL
LIN {X 0,Y 404.604,Z 211.702,A -85,B 0,C 180,E1 -10800,E2 -10800} C_VEL
LIN {X 0,Y 404.415,Z 211.729,A -85,B 0,C 180,E1 -10802.988,E2 -10802.988} C_VEL
LIN {X 0,Y 404.414,Z 211.733,A -85,B 0,C 180,E1 -10805.985,E2 -10805.985} C_VEL
LIN {X 0,Y 404.283,Z 211.748,A -85,B 0,C 180,E1 -10809.001,E2 -10809.001} C_VEL
LIN {X 0,Y 404.248,Z 211.755,A -85,B 0,C 180,E1 -10812.042,E2 -10812.042} C_VEL
LIN {X 0,Y 404.203,Z 211.761,A -85,B 0,C 180,E1 -10815.118,E2 -10815.118} C_VEL
LIN {X 0,Y 404.202,Z 211.758,A -85,B 0,C 180,E1 -10818.238,E2 -10818.238} C_VEL
LIN {X 0,Y 404.13,Z 211.763,A -85,B 0,C 180,E1 -10821.42,E2 -10821.42} C_VEL
LIN {X 0,Y 404.17,Z 211.762,A -85,B 0,C 180,E1 -10824.666,E2 -10824.666} C_VEL
LIN {X 0,Y 404.191,Z 211.765,A -85,B 0,C 180,E1 -10828,E2 -10828} C_VEL
LIN {X 0,Y 404.139,Z 211.768,A -85,B 0,C 180,E1 -10831.56,E2 -10831.56} C_VEL
LIN {X 0,Y 404.178,Z 211.761,A -85,B 0,C 180,E1 -10835.017,E2 -10835.017} C_VEL
LIN {X 0,Y 404.149,Z 211.762,A -85,B 0,C 180,E1 -10838.757,E2 -10838.757} C_VEL
LIN {X 0,Y 404.117,Z 211.76,A -85,B 0,C 180,E1 -10841.6,E2 -10841.6} C_VEL
LIN {X 0,Y 404.14,Z 211.768,A -85,B 0,C 180,E1 -10844.523,E2 -10844.523} C_VEL
LIN {X 0,Y 404.166,Z 211.764,A -85,B 0,C 180,E1 -10847.301,E2 -10847.301} C_VEL
LIN {X 0,Y 404.165,Z 211.764,A -85,B 0,C 180,E1 -10849.956,E2 -10849.956} C_VEL
LIN {X 0,Y 404.137,Z 211.763,A -85,B 0,C 180,E1 -10853.125,E2 -10853.125} C_VEL
LIN {X 0,Y 404.175,Z 211.912,A -85,B 0,C 180,E1 -10856.079,E2 -10856.079} C_VEL
LIN {X 0,Y 408.299,Z 227.76,A -85,B 0,C 180,E1 -10859.389,E2 -10859.389} C_VEL
LIN {X 0,Y 410.858,Z 239.281,A -85,B 0,C 180,E1 -10861.662,E2 -10861.662} C_VEL
LIN {X 0,Y 410.814,Z 241.557,A -85,B 0,C 180,E1 -10862.037,E2 -10862.037} C_VEL
LIN {X 0,Y 416.834,Z 271.28,A -85,B 0,C 180,E1 -10863.035,E2 -10863.035} C_VEL
LIN {X 0,Y 417.868,Z 277.41,A -85,B 0,C 180,E1 -10863.222,E2 -10863.222} C_VEL
LIN {X 0,Y 415.325,Z 405.694,A -85,B 0,C 180,E1 -10865.474,E2 -10865.474} C_VEL
LIN {X 0,Y 414.702,Z 420.881,A -85,B 0,C 180,E1 -10865.901,E2 -10865.901} C_VEL
LIN {X 0,Y 413.81,Z 434.355,A -85,B 0,C 180,E1 -10866.442,E2 -10866.442} C_VEL
LIN {X 0,Y 412.696,Z 448.678,A -85,B 0,C 180,E1 -10867.206,E2 -10867.206} C_VEL
LIN {X 0,Y 411.338,Z 462.985,A -85,B 0,C 180,E1 -10868.185,E2 -10868.185} C_VEL
LIN {X 0,Y 410.039,Z 476.018,A -85,B 0,C 180,E1 -10869.298,E2 -10869.298} C_VEL
LIN {X 0,Y 408.491,Z 489.125,A -85,B 0,C 180,E1 -10870.659,E2 -10870.659} C_VEL
LIN {X 0,Y 407.236,Z 500.997,A -85,B 0,C 180,E1 -10872.162,E2 -10872.162} C_VEL
LIN {X 0,Y 406.009,Z 510.987,A -85,B 0,C 180,E1 -10873.663,E2 -10873.663} C_VEL
LIN {X 0,Y 404.964,Z 520.766,A -85,B 0,C 180,E1 -10875.426,E2 -10875.426} C_VEL
LIN {X 0,Y 404.195,Z 528.931,A -85,B 0,C 180,E1 -10877.192,E2 -10877.192} C_VEL
LIN {X 0,Y 403.655,Z 535.683,A -85,B 0,C 180,E1 -10878.959,E2 -10878.959} C_VEL
LIN {X 0,Y 403.178,Z 541.92,A -85,B 0,C 180,E1 -10880.974,E2 -10880.974} C_VEL
LIN {X 0,Y 402.981,Z 546.748,A -85,B 0,C 180,E1 -10882.988,E2 -10882.988} C_VEL
LIN {X 0,Y 402.851,Z 550.285,A -85,B 0,C 180,E1 -10884.996,E2 -10884.996} C_VEL
LIN {X 0,Y 402.801,Z 552.612,A -85,B 0,C 180,E1 -10887,E2 -10887} C_VEL
LIN {X 0,Y 402.86,Z 553.784,A -85,B 0,C 180,E1 -10889,E2 -10889} C_VEL
LIN {X 0,Y 402.86,Z 553.782,A -85,B 0,C 180,E1 -10891,E2 -10891} C_VEL
LIN {X 0,Y 402.801,Z 552.603,A -85,B 0,C 180,E1 -10893,E2 -10893} C_VEL
LIN {X 0,Y 402.855,Z 550.272,A -85,B 0,C 180,E1 -10895.004,E2 -10895.004} C_VEL
LIN {X 0,Y 402.983,Z 546.737,A -85,B 0,C 180,E1 -10897.012,E2 -10897.012} C_VEL
LIN {X 0,Y 403.178,Z 541.907,A -85,B 0,C 180,E1 -10899.026,E2 -10899.026} C_VEL
LIN {X 0,Y 403.655,Z 535.657,A -85,B 0,C 180,E1 -10901.041,E2 -10901.041} C_VEL
LIN {X 0,Y 404.205,Z 527.807,A -85,B 0,C 180,E1 -10903.063,E2 -10903.063} C_VEL
LIN {X 0,Y 405.122,Z 519.469,A -85,B 0,C 180,E1 -10904.825,E2 -10904.825} C_VEL
LIN {X 0,Y 406.192,Z 509.423,A -85,B 0,C 180,E1 -10906.587,E2 -10906.587} C_VEL
LIN {X 0,Y 407.411,Z 499.155,A -85,B 0,C 180,E1 -10908.089,E2 -10908.089} C_VEL
LIN {X 0,Y 408.808,Z 486.923,A -85,B 0,C 180,E1 -10909.586,E2 -10909.586} C_VEL
LIN {X 0,Y 410.207,Z 474.651,A -85,B 0,C 180,E1 -10910.824,E2 -10910.824} C_VEL
LIN {X 0,Y 411.358,Z 462.883,A -85,B 0,C 180,E1 -10911.814,E2 -10911.814} C_VEL
LIN {X 0,Y 412.696,Z 448.55,A -85,B 0,C 180,E1 -10912.794,E2 -10912.794} C_VEL
LIN {X 0,Y 413.807,Z 434.347,A -85,B 0,C 180,E1 -10913.551,E2 -10913.551} C_VEL
LIN {X 0,Y 414.713,Z 419.744,A -85,B 0,C 180,E1 -10914.131,E2 -10914.131} C_VEL
LIN {X 0,Y 415.372,Z 403.799,A -85,B 0,C 180,E1 -10914.556,E2 -10914.556} C_VEL
LIN {X 0,Y 417.79,Z 278.332,A -85,B 0,C 180,E1 -10916.757,E2 -10916.757} C_VEL
LIN {X 0,Y 417.211,Z 273.692,A -85,B 0,C 180,E1 -10916.884,E2 -10916.884} C_VEL
LIN {X 0,Y 411.403,Z 244.146,A -85,B 0,C 180,E1 -10917.86,E2 -10917.86} C_VEL
LIN {X 0,Y 410.835,Z 241.163,A -85,B 0,C 180,E1 -10917.992,E2 -10917.992} C_VEL
LIN {X 0,Y 410.579,Z 237.65,A -85,B 0,C 180,E1 -10918.638,E2 -10918.638} C_VEL
LIN {X 0,Y 407.577,Z 225.06,A -85,B 0,C 180,E1 -10921.151,E2 -10921.151} C_VEL
LIN {X 0,Y 404.158,Z 211.756,A -85,B 0,C 180,E1 -10923.96,E2 -10923.96} C_VEL
LIN {X 0,Y 404.145,Z 211.769,A -85,B 0,C 180,E1 -10927.49,E2 -10927.49} C_VEL
LIN {X 0,Y 404.162,Z 211.768,A -85,B 0,C 180,E1 -10930.083,E2 -10930.083} C_VEL
LIN {X 0,Y 404.153,Z 211.763,A -85,B 0,C 180,E1 -10933.084,E2 -10933.084} C_VEL
LIN {X 0,Y 404.152,Z 211.762,A -85,B 0,C 180,E1 -10936.915,E2 -10936.915} C_VEL
LIN {X 0,Y 404.163,Z 211.763,A -85,B 0,C 180,E1 -10939.955,E2 -10939.955} C_VEL
LIN {X 0,Y 404.134,Z 211.764,A -85,B 0,C 180,E1 -10943.124,E2 -10943.124} C_VEL
LIN {X 0,Y 404.139,Z 211.764,A -85,B 0,C 180,E1 -10946.187,E2 -10946.187} C_VEL
LIN {X 0,Y 404.148,Z 211.764,A -85,B 0,C 180,E1 -10949.715,E2 -10949.715} C_VEL
LIN {X 0,Y 404.188,Z 211.758,A -85,B 0,C 180,E1 -10953.122,E2 -10953.122} C_VEL
LIN {X 0,Y 404.167,Z 211.765,A -85,B 0,C 180,E1 -10955.334,E2 -10955.334} C_VEL
LIN {X 0,Y 404.13,Z 211.75,A -85,B 0,C 180,E1 -10958.58,E2 -10958.58} C_VEL
LIN {X 0,Y 404.202,Z 211.763,A -85,B 0,C 180,E1 -10961.762,E2 -10961.762} C_VEL
LIN {X 0,Y 404.198,Z 211.758,A -85,B 0,C 180,E1 -10964.882,E2 -10964.882} C_VEL
LIN {X 0,Y 404.249,Z 211.753,A -85,B 0,C 180,E1 -10967.958,E2 -10967.958} C_VEL
LIN {X 0,Y 404.397,Z 211.733,A -85,B 0,C 180,E1 -10972.129,E2 -10972.129} C_VEL
LIN {X 0,Y 404.415,Z 211.732,A -85,B 0,C 180,E1 -10974.015,E2 -10974.015} C_VEL
LIN {X 0,Y 404.474,Z 211.725,A -85,B 0,C 180,E1 -10978.009,E2 -10978.009} C_VEL
LIN {X 0,Y 404.604,Z 211.704,A -85,B 0,C 180,E1 -10980,E2 -10980} C_VEL
LIN {X 0,Y 404.415,Z 211.735,A -85,B 0,C 180,E1 -10982.989,E2 -10982.989} C_VEL
LIN {X 0,Y 404.399,Z 211.737,A -85,B 0,C 180,E1 -10986.988,E2 -10986.988} C_VEL
LIN {X 0,Y 404.251,Z 211.752,A -85,B 0,C 180,E1 -10990.012,E2 -10990.012} C_VEL
LIN {X 0,Y 404.259,Z 211.751,A -85,B 0,C 180,E1 -10993.212,E2 -10993.212} C_VEL
LIN {X 0,Y 404.208,Z 211.757,A -85,B 0,C 180,E1 -10997.007,E2 -10997.007} C_VEL
LIN {X 0,Y 404.156,Z 211.762,A -85,B 0,C 180,E1 -11000.352,E2 -11000.352} C_VEL
LIN {X 0,Y 404.157,Z 211.762,A -85,B 0,C 180,E1 -11003.575,E2 -11003.575} C_VEL
LIN {X 0,Y 404.177,Z 211.741,A -85,B 0,C 180,E1 -11005.767,E2 -11005.767} C_VEL
LIN {X 0,Y 404.192,Z 211.756,A -85,B 0,C 180,E1 -11008,E2 -11008} C_VEL
LIN {X 0,Y 404.137,Z 211.767,A -85,B 0,C 180,E1 -11011.56,E2 -11011.56} C_VEL
LIN {X 0,Y 404.18,Z 211.765,A -85,B 0,C 180,E1 -11015.017,E2 -11015.017} C_VEL
LIN {X 0,Y 404.151,Z 211.766,A -85,B 0,C 180,E1 -11018.757,E2 -11018.757} C_VEL
LIN {X 0,Y 404.119,Z 211.765,A -85,B 0,C 180,E1 -11021.601,E2 -11021.601} C_VEL
LIN {X 0,Y 404.146,Z 211.765,A -85,B 0,C 180,E1 -11024.524,E2 -11024.524} C_VEL
LIN {X 0,Y 404.136,Z 211.769,A -85,B 0,C 180,E1 -11027.297,E2 -11027.297} C_VEL
LIN {X 0,Y 404.166,Z 211.765,A -85,B 0,C 180,E1 -11029.956,E2 -11029.956} C_VEL
LIN {X 0,Y 404.134,Z 211.769,A -85,B 0,C 180,E1 -11033.126,E2 -11033.126} C_VEL
LIN {X 0,Y 404.143,Z 211.767,A -85,B 0,C 180,E1 -11036.188,E2 -11036.188} C_VEL
LIN {X 0,Y 404.177,Z 211.918,A -85,B 0,C 180,E1 -11039.574,E2 -11039.574} C_VEL
LIN {X 0,Y 406.711,Z 221.792,A -85,B 0,C 180,E1 -11041.798,E2 -11041.798} C_VEL
LIN {X 0,Y 415.967,Z 242.735,A -85,B 0,C 180,E1 -11042.885,E2 -11042.885} C_VEL
LIN {X 0,Y 417.378,Z 246.733,A -85,B 0,C 180,E1 -11043.061,E2 -11043.061} C_VEL
LIN {X 0,Y 418.175,Z 250.453,A -85,B 0,C 180,E1 -11043.187,E2 -11043.187} C_VEL
LIN {X 0,Y 415.997,Z 368.146,A -85,B 0,C 180,E1 -11045.25,E2 -11045.25} C_VEL
LIN {X 0,Y 415.503,Z 388.674,A -85,B 0,C 180,E1 -11045.652,E2 -11045.652} C_VEL
LIN {X 0,Y 414.905,Z 403.116,A -85,B 0,C 180,E1 -11046.109,E2 -11046.109} C_VEL
LIN {X 0,Y 414.093,Z 417.07,A -85,B 0,C 180,E1 -11046.728,E2 -11046.728} C_VEL
LIN {X 0,Y 412.88,Z 432.171,A -85,B 0,C 180,E1 -11047.613,E2 -11047.613} C_VEL
LIN {X 0,Y 411.726,Z 445.421,A -85,B 0,C 180,E1 -11048.601,E2 -11048.601} C_VEL
LIN {X 0,Y 410.269,Z 458.888,A -85,B 0,C 180,E1 -11049.834,E2 -11049.834} C_VEL
LIN {X 0,Y 408.927,Z 471.213,A -85,B 0,C 180,E1 -11051.217,E2 -11051.217} C_VEL
LIN {X 0,Y 407.603,Z 482.22,A -85,B 0,C 180,E1 -11052.697,E2 -11052.697} C_VEL
LIN {X 0,Y 406.347,Z 493.019,A -85,B 0,C 180,E1 -11054.45,E2 -11054.45} C_VEL
LIN {X 0,Y 405.2,Z 502.263,A -85,B 0,C 180,E1 -11056.267,E2 -11056.267} C_VEL
LIN {X 0,Y 404.584,Z 509.398,A -85,B 0,C 180,E1 -11057.969,E2 -11057.969} C_VEL
LIN {X 0,Y 403.808,Z 516.338,A -85,B 0,C 180,E1 -11059.977,E2 -11059.977} C_VEL
LIN {X 0,Y 403.77,Z 516.725,A -85,B 0,C 180,E1 -11060.108,E2 -11060.108} C_VEL
LIN {X 0,Y 402.912,Z 519.016,A -85,B 0,C 180,E1 -11060.875,E2 -11060.875} C_VEL
LIN {X 0,Y 399.808,Z 522.409,A -85,B 0,C 180,E1 -11062.131,E2 -11062.131} C_VEL
LIN {X 0,Y 397.248,Z 524.743,A -85,B 0,C 180,E1 -11063.163,E2 -11063.163} C_VEL
LIN {X 0,Y 396.122,Z 526.249,A -85,B 0,C 180,E1 -11063.975,E2 -11063.975} C_VEL
LIN {X 0,Y 396.013,Z 526.672,A -85,B 0,C 180,E1 -11064.253,E2 -11064.253} C_VEL
LIN {X 0,Y 395.826,Z 528.995,A -85,B 0,C 180,E1 -11065.927,E2 -11065.927} C_VEL
LIN {X 0,Y 395.836,Z 530.732,A -85,B 0,C 180,E1 -11067.965,E2 -11067.965} C_VEL
LIN {X 0,Y 395.777,Z 531.341,A -85,B 0,C 180,E1 -11070,E2 -11070} C_VEL
LIN {X 0,Y 395.836,Z 530.78,A -85,B 0,C 180,E1 -11072.035,E2 -11072.035} C_VEL
LIN {X 0,Y 395.825,Z 529.106,A -85,B 0,C 180,E1 -11074.073,E2 -11074.073} C_VEL
LIN {X 0,Y 396.031,Z 526.274,A -85,B 0,C 180,E1 -11076.112,E2 -11076.112} C_VEL
LIN {X 0,Y 396.314,Z 522.22,A -85,B 0,C 180,E1 -11078.156,E2 -11078.156} C_VEL
LIN {X 0,Y 396.773,Z 516.843,A -85,B 0,C 180,E1 -11080.202,E2 -11080.202} C_VEL
LIN {X 0,Y 397.609,Z 509.985,A -85,B 0,C 180,E1 -11082.246,E2 -11082.246} C_VEL
LIN {X 0,Y 398.224,Z 503.171,A -85,B 0,C 180,E1 -11083.913,E2 -11083.913} C_VEL
LIN {X 0,Y 399.222,Z 495.073,A -85,B 0,C 180,E1 -11085.573,E2 -11085.573} C_VEL
LIN {X 0,Y 400.528,Z 484.664,A -85,B 0,C 180,E1 -11087.355,E2 -11087.355} C_VEL
LIN {X 0,Y 401.907,Z 473.504,A -85,B 0,C 180,E1 -11088.938,E2 -11088.938} C_VEL
LIN {X 0,Y 403.361,Z 461.122,A -85,B 0,C 180,E1 -11090.393,E2 -11090.393} C_VEL
LIN {X 0,Y 404.831,Z 448.113,A -85,B 0,C 180,E1 -11091.648,E2 -11091.648} C_VEL
LIN {X 0,Y 406.08,Z 435.449,A -85,B 0,C 180,E1 -11092.648,E2 -11092.648} C_VEL
LIN {X 0,Y 407.352,Z 420.949,A -85,B 0,C 180,E1 -11093.56,E2 -11093.56} C_VEL
LIN {X 0,Y 408.274,Z 405.536,A -85,B 0,C 180,E1 -11094.304,E2 -11094.304} C_VEL
LIN {X 0,Y 408.987,Z 391.097,A -85,B 0,C 180,E1 -11094.796,E2 -11094.796} C_VEL
LIN {X 0,Y 409.509,Z 371.841,A -85,B 0,C 180,E1 -11095.203,E2 -11095.203} C_VEL
LIN {X 0,Y 411.299,Z 282.857,A -85,B 0,C 180,E1 -11096.779,E2 -11096.779} C_VEL
LIN {X 0,Y 411.765,Z 251.033,A -85,B 0,C 180,E1 -11097.358,E2 -11097.358} C_VEL
LIN {X 0,Y 410.531,Z 246.795,A -85,B 0,C 180,E1 -11097.53,E2 -11097.53} C_VEL
LIN {X 0,Y 402.223,Z 227.816,A -85,B 0,C 180,E1 -11098.531,E2 -11098.531} C_VEL
LIN {X 0,Y 399.452,Z 221.626,A -85,B 0,C 180,E1 -11098.902,E2 -11098.902} C_VEL
LIN {X 0,Y 397.122,Z 212.647,A -85,B 0,C 180,E1 -11101.026,E2 -11101.026} C_VEL
LIN {X 0,Y 397.124,Z 212.643,A -85,B 0,C 180,E1 -11104.492,E2 -11104.492} C_VEL
LIN {X 0,Y 397.103,Z 212.648,A -85,B 0,C 180,E1 -11108.274,E2 -11108.274} C_VEL
LIN {X 0,Y 397.086,Z 212.646,A -85,B 0,C 180,E1 -11110.908,E2 -11110.908} C_VEL
LIN {X 0,Y 397.1,Z 212.646,A -85,B 0,C 180,E1 -11113.647,E2 -11113.647} C_VEL
LIN {X 0,Y 397.1,Z 212.643,A -85,B 0,C 180,E1 -11116.52,E2 -11116.52} C_VEL
LIN {X 0,Y 397.115,Z 212.645,A -85,B 0,C 180,E1 -11119.551,E2 -11119.551} C_VEL
LIN {X 0,Y 397.093,Z 212.631,A -85,B 0,C 180,E1 -11122.789,E2 -11122.789} C_VEL
LIN {X 0,Y 397.113,Z 212.641,A -85,B 0,C 180,E1 -11126.281,E2 -11126.281} C_VEL
LIN {X 0,Y 397.108,Z 212.636,A -85,B 0,C 180,E1 -11130.133,E2 -11130.133} C_VEL
LIN {X 0,Y 397.188,Z 212.635,A -85,B 0,C 180,E1 -11132.609,E2 -11132.609} C_VEL
LIN {X 0,Y 397.126,Z 212.64,A -85,B 0,C 180,E1 -11135.981,E2 -11135.981} C_VEL
LIN {X 0,Y 397.131,Z 212.639,A -85,B 0,C 180,E1 -11139.704,E2 -11139.704} C_VEL
LIN {X 0,Y 397.174,Z 212.635,A -85,B 0,C 180,E1 -11142.844,E2 -11142.844} C_VEL
LIN {X 0,Y 397.221,Z 212.626,A -85,B 0,C 180,E1 -11146.702,E2 -11146.702} C_VEL
LIN {X 0,Y 397.21,Z 212.624,A -85,B 0,C 180,E1 -11149.809,E2 -11149.809} C_VEL
LIN {X 0,Y 397.344,Z 212.616,A -85,B 0,C 180,E1 -11152.888,E2 -11152.888} C_VEL
LIN {X 0,Y 397.247,Z 212.622,A -85,B 0,C 180,E1 -11154.925,E2 -11154.925} C_VEL
LIN {X 0,Y 397.443,Z 212.6,A -85,B 0,C 180,E1 -11157.973,E2 -11157.973} C_VEL
LIN {X 0,Y 397.574,Z 212.578,A -85,B 0,C 180,E1 -11160,E2 -11160} C_VEL
LIN {X 0,Y 397.373,Z 212.606,A -85,B 0,C 180,E1 -11163.041,E2 -11163.041} C_VEL
LIN {X 0,Y 397.365,Z 212.611,A -85,B 0,C 180,E1 -11166.092,E2 -11166.092} C_VEL
LIN {X 0,Y 397.245,Z 212.624,A -85,B 0,C 180,E1 -11169.162,E2 -11169.162} C_VEL
LIN {X 0,Y 397.211,Z 212.631,A -85,B 0,C 180,E1 -11172.258,E2 -11172.258} C_VEL
LIN {X 0,Y 397.176,Z 212.636,A -85,B 0,C 180,E1 -11175.392,E2 -11175.392} C_VEL
LIN {X 0,Y 397.154,Z 212.641,A -85,B 0,C 180,E1 -11178.574,E2 -11178.574} C_VEL
LIN {X 0,Y 397.089,Z 212.642,A -85,B 0,C 180,E1 -11181.819,E2 -11181.819} C_VEL
LIN {X 0,Y 397.149,Z 212.634,A -85,B 0,C 180,E1 -11185.132,E2 -11185.132} C_VEL
LIN {X 0,Y 397.156,Z 212.639,A -85,B 0,C 180,E1 -11187.777,E2 -11187.777} C_VEL
LIN {X 0,Y 397.079,Z 212.647,A -85,B 0,C 180,E1 -11190.882,E2 -11190.882} C_VEL
LIN {X 0,Y 397.119,Z 212.644,A -85,B 0,C 180,E1 -11194.494,E2 -11194.494} C_VEL
LIN {X 0,Y 397.096,Z 212.645,A -85,B 0,C 180,E1 -11198.276,E2 -11198.276} C_VEL
LIN {X 0,Y 397.083,Z 212.63,A -85,B 0,C 180,E1 -11200.909,E2 -11200.909} C_VEL
LIN {X 0,Y 397.096,Z 212.648,A -85,B 0,C 180,E1 -11203.649,E2 -11203.649} C_VEL
LIN {X 0,Y 397.099,Z 212.644,A -85,B 0,C 180,E1 -11206.521,E2 -11206.521} C_VEL
LIN {X 0,Y 397.116,Z 212.644,A -85,B 0,C 180,E1 -11209.552,E2 -11209.552} C_VEL
LIN {X 0,Y 397.095,Z 212.637,A -85,B 0,C 180,E1 -11212.791,E2 -11212.791} C_VEL
LIN {X 0,Y 397.123,Z 212.656,A -85,B 0,C 180,E1 -11215.579,E2 -11215.579} C_VEL
LIN {X 0,Y 401.03,Z 227.589,A -85,B 0,C 180,E1 -11218.782,E2 -11218.782} C_VEL
LIN {X 0,Y 404.069,Z 241.077,A -85,B 0,C 180,E1 -11221.508,E2 -11221.508} C_VEL
LIN {X 0,Y 408.501,Z 261.837,A -85,B 0,C 180,E1 -11222.26,E2 -11222.26} C_VEL
LIN {X 0,Y 411.504,Z 278.124,A -85,B 0,C 180,E1 -11222.791,E2 -11222.791} C_VEL
LIN {X 0,Y 408.888,Z 405.51,A -85,B 0,C 180,E1 -11225.062,E2 -11225.062} C_VEL
LIN {X 0,Y 408.242,Z 420.69,A -85,B 0,C 180,E1 -11225.495,E2 -11225.495} C_VEL
LIN {X 0,Y 407.337,Z 433.941,A -85,B 0,C 180,E1 -11226.033,E2 -11226.033} C_VEL
LIN {X 0,Y 406.144,Z 448.482,A -85,B 0,C 180,E1 -11226.818,E2 -11226.818} C_VEL
LIN {X 0,Y 404.728,Z 462.788,A -85,B 0,C 180,E1 -11227.81,E2 -11227.81} C_VEL
LIN {X 0,Y 403.313,Z 475.817,A -85,B 0,C 180,E1 -11228.937,E2 -11228.937} C_VEL
LIN {X 0,Y 401.888,Z 487.852,A -85,B 0,C 180,E1 -11230.196,E2 -11230.196} C_VEL
LIN {X 0,Y 400.595,Z 499.004,A -85,B 0,C 180,E1 -11231.592,E2 -11231.592} C_VEL
LIN {X 0,Y 399.335,Z 509.267,A -85,B 0,C 180,E1 -11233.119,E2 -11233.119} C_VEL
LIN {X 0,Y 398.178,Z 519.304,A -85,B 0,C 180,E1 -11234.91,E2 -11234.91} C_VEL
LIN {X 0,Y 397.151,Z 528.453,A -85,B 0,C 180,E1 -11236.891,E2 -11236.891} C_VEL
LIN {X 0,Y 396.616,Z 535.481,A -85,B 0,C 180,E1 -11238.76,E2 -11238.76} C_VEL
LIN {X 0,Y 396.094,Z 541.718,A -85,B 0,C 180,E1 -11240.811,E2 -11240.811} C_VEL
LIN {X 0,Y 395.905,Z 546.547,A -85,B 0,C 180,E1 -11242.862,E2 -11242.862} C_VEL
LIN {X 0,Y 395.752,Z 550.083,A -85,B 0,C 180,E1 -11244.906,E2 -11244.906} C_VEL
LIN {X 0,Y 395.703,Z 552.411,A -85,B 0,C 180,E1 -11246.946,E2 -11246.946} C_VEL
LIN {X 0,Y 395.788,Z 553.584,A -85,B 0,C 180,E1 -11248.983,E2 -11248.983} C_VEL
LIN {X 0,Y 395.788,Z 553.582,A -85,B 0,C 180,E1 -11251.017,E2 -11251.017} C_VEL
LIN {X 0,Y 395.703,Z 552.402,A -85,B 0,C 180,E1 -11253.054,E2 -11253.054} C_VEL
LIN {X 0,Y 395.755,Z 550.07,A -85,B 0,C 180,E1 -11255.094,E2 -11255.094} C_VEL
LIN {X 0,Y 395.906,Z 546.534,A -85,B 0,C 180,E1 -11257.138,E2 -11257.138} C_VEL
LIN {X 0,Y 396.094,Z 541.703,A -85,B 0,C 180,E1 -11259.189,E2 -11259.189} C_VEL
LIN {X 0,Y 396.615,Z 535.453,A -85,B 0,C 180,E1 -11261.24,E2 -11261.24} C_VEL
LIN {X 0,Y 397.19,Z 527.602,A -85,B 0,C 180,E1 -11263.298,E2 -11263.298} C_VEL
LIN {X 0,Y 398.18,Z 519.263,A -85,B 0,C 180,E1 -11265.09,E2 -11265.09} C_VEL
LIN {X 0,Y 399.339,Z 509.218,A -85,B 0,C 180,E1 -11266.881,E2 -11266.881} C_VEL
LIN {X 0,Y 400.571,Z 498.949,A -85,B 0,C 180,E1 -11268.409,E2 -11268.409} C_VEL
LIN {X 0,Y 402.073,Z 486.718,A -85,B 0,C 180,E1 -11269.928,E2 -11269.928} C_VEL
LIN {X 0,Y 403.631,Z 473.104,A -85,B 0,C 180,E1 -11271.313,E2 -11271.313} C_VEL
LIN {X 0,Y 405.062,Z 459.457,A -85,B 0,C 180,E1 -11272.439,E2 -11272.439} C_VEL
LIN {X 0,Y 406.441,Z 445.326,A -85,B 0,C 180,E1 -11273.367,E2 -11273.367} C_VEL
LIN {X 0,Y 407.584,Z 430.068,A -85,B 0,C 180,E1 -11274.14,E2 -11274.14} C_VEL
LIN {X 0,Y 408.476,Z 414.84,A -85,B 0,C 180,E1 -11274.693,E2 -11274.693} C_VEL
LIN {X 0,Y 409.063,Z 398.871,A -85,B 0,C 180,E1 -11275.062,E2 -11275.062} C_VEL
LIN {X 0,Y 411.432,Z 278.393,A -85,B 0,C 180,E1 -11277.199,E2 -11277.199} C_VEL
LIN {X 0,Y 406.736,Z 253.094,A -85,B 0,C 180,E1 -11278.029,E2 -11278.029} C_VEL
LIN {X 0,Y 404.094,Z 241.089,A -85,B 0,C 180,E1 -11278.476,E2 -11278.476} C_VEL
LIN {X 0,Y 401.347,Z 229.062,A -85,B 0,C 180,E1 -11280.903,E2 -11280.903} C_VEL
LIN {X 0,Y 397.758,Z 215.173,A -85,B 0,C 180,E1 -11283.856,E2 -11283.856} C_VEL
LIN {X 0,Y 397.128,Z 212.638,A -85,B 0,C 180,E1 -11284.441,E2 -11284.441} C_VEL
LIN {X 0,Y 397.105,Z 212.647,A -85,B 0,C 180,E1 -11288.274,E2 -11288.274} C_VEL
LIN {X 0,Y 397.108,Z 212.643,A -85,B 0,C 180,E1 -11290.905,E2 -11290.905} C_VEL
LIN {X 0,Y 397.098,Z 212.645,A -85,B 0,C 180,E1 -11293.648,E2 -11293.648} C_VEL
LIN {X 0,Y 397.099,Z 212.642,A -85,B 0,C 180,E1 -11296.52,E2 -11296.52} C_VEL
LIN {X 0,Y 397.114,Z 212.639,A -85,B 0,C 180,E1 -11299.551,E2 -11299.551} C_VEL
LIN {X 0,Y 397.092,Z 212.641,A -85,B 0,C 180,E1 -11302.79,E2 -11302.79} C_VEL
LIN {X 0,Y 397.112,Z 212.638,A -85,B 0,C 180,E1 -11306.282,E2 -11306.282} C_VEL
LIN {X 0,Y 397.08,Z 212.644,A -85,B 0,C 180,E1 -11309.118,E2 -11309.118} C_VEL
LIN {X 0,Y 397.188,Z 212.629,A -85,B 0,C 180,E1 -11312.609,E2 -11312.609} C_VEL
LIN {X 0,Y 397.121,Z 212.638,A -85,B 0,C 180,E1 -11315.981,E2 -11315.981} C_VEL
LIN {X 0,Y 397.131,Z 212.629,A -85,B 0,C 180,E1 -11319.704,E2 -11319.704} C_VEL
LIN {X 0,Y 397.174,Z 212.633,A -85,B 0,C 180,E1 -11322.845,E2 -11322.845} C_VEL
LIN {X 0,Y 397.221,Z 212.627,A -85,B 0,C 180,E1 -11326.703,E2 -11326.703} C_VEL
LIN {X 0,Y 397.21,Z 212.632,A -85,B 0,C 180,E1 -11329.809,E2 -11329.809} C_VEL
LIN {X 0,Y 397.344,Z 212.611,A -85,B 0,C 180,E1 -11332.888,E2 -11332.888} C_VEL
LIN {X 0,Y 397.247,Z 212.625,A -85,B 0,C 180,E1 -11334.925,E2 -11334.925} C_VEL
LIN {X 0,Y 397.443,Z 212.601,A -85,B 0,C 180,E1 -11337.973,E2 -11337.973} C_VEL
LIN {X 0,Y 397.574,Z 212.58,A -85,B 0,C 180,E1 -11340,E2 -11340} C_VEL
LIN {X 0,Y 397.374,Z 212.613,A -85,B 0,C 180,E1 -11343.042,E2 -11343.042} C_VEL
LIN {X 0,Y 397.342,Z 212.614,A -85,B 0,C 180,E1 -11346.655,E2 -11346.655} C_VEL
LIN {X 0,Y 397.245,Z 212.623,A -85,B 0,C 180,E1 -11349.162,E2 -11349.162} C_VEL
LIN {X 0,Y 397.212,Z 212.626,A -85,B 0,C 180,E1 -11352.258,E2 -11352.258} C_VEL
LIN {X 0,Y 397.173,Z 212.636,A -85,B 0,C 180,E1 -11355.392,E2 -11355.392} C_VEL
LIN {X 0,Y 397.155,Z 212.637,A -85,B 0,C 180,E1 -11358.574,E2 -11358.574} C_VEL
LIN {X 0,Y 397.088,Z 212.645,A -85,B 0,C 180,E1 -11361.819,E2 -11361.819} C_VEL
LIN {X 0,Y 397.146,Z 212.618,A -85,B 0,C 180,E1 -11365.513,E2 -11365.513} C_VEL
LIN {X 0,Y 397.121,Z 212.639,A -85,B 0,C 180,E1 -11368.544,E2 -11368.544} C_VEL
LIN {X 0,Y 397.075,Z 212.646,A -85,B 0,C 180,E1 -11372.072,E2 -11372.072} C_VEL
LIN {X 0,Y 397.115,Z 212.641,A -85,B 0,C 180,E1 -11375.504,E2 -11375.504} C_VEL
LIN {X 0,Y 397.126,Z 212.64,A -85,B 0,C 180,E1 -11378.862,E2 -11378.862} C_VEL
LIN {X 0,Y 397.066,Z 212.644,A -85,B 0,C 180,E1 -11382.268,E2 -11382.268} C_VEL
LIN {X 0,Y 397.089,Z 212.648,A -85,B 0,C 180,E1 -11385.069,E2 -11385.069} C_VEL
LIN {X 0,Y 397.065,Z 212.649,A -85,B 0,C 180,E1 -11388.022,E2 -11388.022} C_VEL
LIN {X 0,Y 397.129,Z 212.636,A -85,B 0,C 180,E1 -11391.139,E2 -11391.139} C_VEL
LIN {X 0,Y 397.117,Z 212.639,A -85,B 0,C 180,E1 -11394.497,E2 -11394.497} C_VEL
LIN {X 0,Y 397.077,Z 212.651,A -85,B 0,C 180,E1 -11397.929,E2 -11397.929} C_VEL
LIN {X 0,Y 397.141,Z 212.807,A -85,B 0,C 180,E1 -11399.124,E2 -11399.124} C_VEL
LIN {X 0,Y 399.563,Z 222.025,A -85,B 0,C 180,E1 -11401.246,E2 -11401.246} C_VEL
LIN {X 0,Y 408.015,Z 240.799,A -85,B 0,C 180,E1 -11402.269,E2 -11402.269} C_VEL
LIN {X 0,Y 411.343,Z 249.312,A -85,B 0,C 180,E1 -11402.679,E2 -11402.679} C_VEL
LIN {X 0,Y 411.866,Z 253.068,A -85,B 0,C 180,E1 -11402.789,E2 -11402.789} C_VEL
LIN {X 0,Y 409.457,Z 373.732,A -85,B 0,C 180,E1 -11404.93,E2 -11404.93} C_VEL
LIN {X 0,Y 408.944,Z 391.171,A -85,B 0,C 180,E1 -11405.303,E2 -11405.303} C_VEL
LIN {X 0,Y 408.281,Z 406.038,A -85,B 0,C 180,E1 -11405.818,E2 -11405.818} C_VEL
LIN {X 0,Y 407.451,Z 418.827,A -85,B 0,C 180,E1 -11406.418,E2 -11406.418} C_VEL
LIN {X 0,Y 406.33,Z 432.378,A -85,B 0,C 180,E1 -11407.232,E2 -11407.232} C_VEL
LIN {X 0,Y 405.107,Z 445.628,A -85,B 0,C 180,E1 -11408.234,E2 -11408.234} C_VEL
LIN {X 0,Y 403.585,Z 459.094,A -85,B 0,C 180,E1 -11409.485,E2 -11409.485} C_VEL
LIN {X 0,Y 402.236,Z 470.826,A -85,B 0,C 180,E1 -11410.815,E2 -11410.815} C_VEL
LIN {X 0,Y 400.809,Z 482.425,A -85,B 0,C 180,E1 -11412.394,E2 -11412.394} C_VEL
LIN {X 0,Y 399.48,Z 493.223,A -85,B 0,C 180,E1 -11414.176,E2 -11414.176} C_VEL
LIN {X 0,Y 398.229,Z 502.737,A -85,B 0,C 180,E1 -11416.084,E2 -11416.084} C_VEL
LIN {X 0,Y 397.613,Z 509.601,A -85,B 0,C 180,E1 -11417.755,E2 -11417.755} C_VEL
LIN {X 0,Y 396.794,Z 516.541,A -85,B 0,C 180,E1 -11419.798,E2 -11419.798} C_VEL
LIN {X 0,Y 396.353,Z 521.989,A -85,B 0,C 180,E1 -11421.845,E2 -11421.845} C_VEL
LIN {X 0,Y 396.057,Z 526.103,A -85,B 0,C 180,E1 -11423.888,E2 -11423.888} C_VEL
LIN {X 0,Y 396.013,Z 526.672,A -85,B 0,C 180,E1 -11424.253,E2 -11424.253} C_VEL
LIN {X 0,Y 395.273,Z 527.984,A -85,B 0,C 180,E1 -11425.082,E2 -11425.082} C_VEL
LIN {X 0,Y 392.307,Z 529.684,A -85,B 0,C 180,E1 -11426.436,E2 -11426.436} C_VEL
LIN {X 0,Y 389.84,Z 530.663,A -85,B 0,C 180,E1 -11427.538,E2 -11427.538} C_VEL
LIN {X 0,Y 388.795,Z 531.145,A -85,B 0,C 180,E1 -11428.396,E2 -11428.396} C_VEL
LIN {X 0,Y 388.716,Z 531.263,A -85,B 0,C 180,E1 -11428.686,E2 -11428.686} C_VEL
LIN {X 0,Y 388.706,Z 531.542,A -85,B 0,C 180,E1 -11430,E2 -11430} C_VEL
LIN {X 0,Y 388.738,Z 530.981,A -85,B 0,C 180,E1 -11432.072,E2 -11432.072} C_VEL
LIN {X 0,Y 388.752,Z 529.306,A -85,B 0,C 180,E1 -11434.147,E2 -11434.147} C_VEL
LIN {X 0,Y 388.962,Z 526.474,A -85,B 0,C 180,E1 -11436.224,E2 -11436.224} C_VEL
LIN {X 0,Y 389.262,Z 522.42,A -85,B 0,C 180,E1 -11438.305,E2 -11438.305} C_VEL
LIN {X 0,Y 389.762,Z 517.043,A -85,B 0,C 180,E1 -11440.388,E2 -11440.388} C_VEL
LIN {X 0,Y 390.626,Z 510.185,A -85,B 0,C 180,E1 -11442.468,E2 -11442.468} C_VEL
LIN {X 0,Y 391.31,Z 503.304,A -85,B 0,C 180,E1 -11444.18,E2 -11444.18} C_VEL
LIN {X 0,Y 392.536,Z 493.928,A -85,B 0,C 180,E1 -11446.111,E2 -11446.111} C_VEL
LIN {X 0,Y 393.706,Z 484.864,A -85,B 0,C 180,E1 -11447.665,E2 -11447.665} C_VEL
LIN {X 0,Y 395.125,Z 474.074,A -85,B 0,C 180,E1 -11449.224,E2 -11449.224} C_VEL
LIN {X 0,Y 396.571,Z 462.487,A -85,B 0,C 180,E1 -11450.623,E2 -11450.623} C_VEL
LIN {X 0,Y 398.083,Z 449.728,A -85,B 0,C 180,E1 -11451.897,E2 -11451.897} C_VEL
LIN {X 0,Y 399.36,Z 437.404,A -85,B 0,C 180,E1 -11452.914,E2 -11452.914} C_VEL
LIN {X 0,Y 400.545,Z 424.178,A -85,B 0,C 180,E1 -11453.8,E2 -11453.8} C_VEL
LIN {X 0,Y 401.635,Z 408.799,A -85,B 0,C 180,E1 -11454.593,E2 -11454.593} C_VEL
LIN {X 0,Y 402.461,Z 393.558,A -85,B 0,C 180,E1 -11455.157,E2 -11455.157} C_VEL
LIN {X 0,Y 403.006,Z 377.377,A -85,B 0,C 180,E1 -11455.535,E2 -11455.535} C_VEL
LIN {X 0,Y 405.028,Z 279.874,A -85,B 0,C 180,E1 -11457.29,E2 -11457.29} C_VEL
LIN {X 0,Y 405.546,Z 252.562,A -85,B 0,C 180,E1 -11457.787,E2 -11457.787} C_VEL
LIN {X 0,Y 403.798,Z 247.642,A -85,B 0,C 180,E1 -11458.016,E2 -11458.016} C_VEL
LIN {X 0,Y 395.406,Z 228.7,A -85,B 0,C 180,E1 -11459.055,E2 -11459.055} C_VEL
LIN {X 0,Y 392.176,Z 221.867,A -85,B 0,C 180,E1 -11459.486,E2 -11459.486} C_VEL
LIN {X 0,Y 390.048,Z 213.527,A -85,B 0,C 180,E1 -11461.501,E2 -11461.501} C_VEL
LIN {X 0,Y 390.084,Z 213.525,A -85,B 0,C 180,E1 -11465.206,E2 -11465.206} C_VEL
LIN {X 0,Y 390.089,Z 213.517,A -85,B 0,C 180,E1 -11469.091,E2 -11469.091} C_VEL
LIN {X 0,Y 390.041,Z 213.523,A -85,B 0,C 180,E1 -11472.374,E2 -11472.374} C_VEL
LIN {X 0,Y 390.042,Z 213.528,A -85,B 0,C 180,E1 -11475.354,E2 -11475.354} C_VEL
LIN {X 0,Y 390.046,Z 213.515,A -85,B 0,C 180,E1 -11478.188,E2 -11478.188} C_VEL
LIN {X 0,Y 390.09,Z 213.517,A -85,B 0,C 180,E1 -11480.907,E2 -11480.907} C_VEL
LIN {X 0,Y 390.08,Z 213.518,A -85,B 0,C 180,E1 -11484.792,E2 -11484.792} C_VEL
LIN {X 0,Y 390.021,Z 213.507,A -85,B 0,C 180,E1 -11488.495,E2 -11488.495} C_VEL
LIN {X 0,Y 390.111,Z 213.514,A -85,B 0,C 180,E1 -11492.069,E2 -11492.069} C_VEL
LIN {X 0,Y 390.073,Z 213.52,A -85,B 0,C 180,E1 -11495.519,E2 -11495.519} C_VEL
LIN {X 0,Y 390.048,Z 213.524,A -85,B 0,C 180,E1 -11498.877,E2 -11498.877} C_VEL
LIN {X 0,Y 390.12,Z 213.508,A -85,B 0,C 180,E1 -11502.166,E2 -11502.166} C_VEL
LIN {X 0,Y 390.136,Z 213.504,A -85,B 0,C 180,E1 -11505.392,E2 -11505.392} C_VEL
LIN {X 0,Y 390.141,Z 213.514,A -85,B 0,C 180,E1 -11508.571,E2 -11508.571} C_VEL
LIN {X 0,Y 390.3,Z 213.49,A -85,B 0,C 180,E1 -11512.031,E2 -11512.031} C_VEL
LIN {X 0,Y 390.219,Z 213.497,A -85,B 0,C 180,E1 -11514.833,E2 -11514.833} C_VEL
LIN {X 0,Y 390.412,Z 213.476,A -85,B 0,C 180,E1 -11517.937,E2 -11517.937} C_VEL
LIN {X 0,Y 390.543,Z 213.454,A -85,B 0,C 180,E1 -11520,E2 -11520} C_VEL
LIN {X 0,Y 390.307,Z 213.485,A -85,B 0,C 180,E1 -11523.096,E2 -11523.096} C_VEL
LIN {X 0,Y 390.319,Z 213.49,A -85,B 0,C 180,E1 -11526.202,E2 -11526.202} C_VEL
LIN {X 0,Y 390.197,Z 213.502,A -85,B 0,C 180,E1 -11529.329,E2 -11529.329} C_VEL
LIN {X 0,Y 390.186,Z 213.501,A -85,B 0,C 180,E1 -11533.439,E2 -11533.439} C_VEL
LIN {X 0,Y 390.142,Z 213.504,A -85,B 0,C 180,E1 -11537.309,E2 -11537.309} C_VEL
LIN {X 0,Y 390.079,Z 213.52,A -85,B 0,C 180,E1 -11540.47,E2 -11540.47} C_VEL
LIN {X 0,Y 390.082,Z 213.519,A -85,B 0,C 180,E1 -11543.351,E2 -11543.351} C_VEL
LIN {X 0,Y 390.106,Z 213.518,A -85,B 0,C 180,E1 -11546.769,E2 -11546.769} C_VEL
LIN {X 0,Y 390.038,Z 213.527,A -85,B 0,C 180,E1 -11550.3,E2 -11550.3} C_VEL
LIN {X 0,Y 390.049,Z 213.518,A -85,B 0,C 180,E1 -11552.721,E2 -11552.721} C_VEL
LIN {X 0,Y 390.05,Z 213.522,A -85,B 0,C 180,E1 -11555.826,E2 -11555.826} C_VEL
LIN {X 0,Y 390.064,Z 213.516,A -85,B 0,C 180,E1 -11559.219,E2 -11559.219} C_VEL
LIN {X 0,Y 390.037,Z 213.523,A -85,B 0,C 180,E1 -11562.375,E2 -11562.375} C_VEL
LIN {X 0,Y 390.039,Z 213.525,A -85,B 0,C 180,E1 -11565.355,E2 -11565.355} C_VEL
LIN {X 0,Y 390.064,Z 213.52,A -85,B 0,C 180,E1 -11568.192,E2 -11568.192} C_VEL
LIN {X 0,Y 390.091,Z 213.517,A -85,B 0,C 180,E1 -11570.909,E2 -11570.909} C_VEL
LIN {X 0,Y 390.088,Z 213.521,A -85,B 0,C 180,E1 -11575.016,E2 -11575.016} C_VEL
LIN {X 0,Y 390.075,Z 213.548,A -85,B 0,C 180,E1 -11575.088,E2 -11575.088} C_VEL
LIN {X 0,Y 393.832,Z 227.847,A -85,B 0,C 180,E1 -11578.237,E2 -11578.237} C_VEL
LIN {X 0,Y 396.931,Z 241.016,A -85,B 0,C 180,E1 -11580.965,E2 -11580.965} C_VEL
LIN {X 0,Y 398.724,Z 246.154,A -85,B 0,C 180,E1 -11581.21,E2 -11581.21} C_VEL
LIN {X 0,Y 404.558,Z 275.538,A -85,B 0,C 180,E1 -11582.238,E2 -11582.238} C_VEL
LIN {X 0,Y 405.151,Z 279.982,A -85,B 0,C 180,E1 -11582.368,E2 -11582.368} C_VEL
LIN {X 0,Y 402.454,Z 405.325,A -85,B 0,C 180,E1 -11584.636,E2 -11584.636} C_VEL
LIN {X 0,Y 401.79,Z 420.499,A -85,B 0,C 180,E1 -11585.075,E2 -11585.075} C_VEL
LIN {X 0,Y 400.876,Z 433.073,A -85,B 0,C 180,E1 -11585.586,E2 -11585.586} C_VEL
LIN {X 0,Y 399.807,Z 446.293,A -85,B 0,C 180,E1 -11586.291,E2 -11586.291} C_VEL
LIN {X 0,Y 398.297,Z 461.004,A -85,B 0,C 180,E1 -11587.296,E2 -11587.296} C_VEL
LIN {X 0,Y 396.813,Z 474.324,A -85,B 0,C 180,E1 -11588.439,E2 -11588.439} C_VEL
LIN {X 0,Y 395.308,Z 486.578,A -85,B 0,C 180,E1 -11589.716,E2 -11589.716} C_VEL
LIN {X 0,Y 393.745,Z 498.802,A -85,B 0,C 180,E1 -11591.26,E2 -11591.26} C_VEL
LIN {X 0,Y 392.469,Z 509.066,A -85,B 0,C 180,E1 -11592.815,E2 -11592.815} C_VEL
LIN {X 0,Y 391.26,Z 519.103,A -85,B 0,C 180,E1 -11594.637,E2 -11594.637} C_VEL
LIN {X 0,Y 390.215,Z 527.818,A -85,B 0,C 180,E1 -11596.549,E2 -11596.549} C_VEL
LIN {X 0,Y 389.587,Z 535.28,A -85,B 0,C 180,E1 -11598.555,E2 -11598.555} C_VEL
LIN {X 0,Y 389.026,Z 541.516,A -85,B 0,C 180,E1 -11600.643,E2 -11600.643} C_VEL
LIN {X 0,Y 388.824,Z 546.346,A -85,B 0,C 180,E1 -11602.731,E2 -11602.731} C_VEL
LIN {X 0,Y 388.658,Z 549.883,A -85,B 0,C 180,E1 -11604.813,E2 -11604.813} C_VEL
LIN {X 0,Y 388.61,Z 552.21,A -85,B 0,C 180,E1 -11606.89,E2 -11606.89} C_VEL
LIN {X 0,Y 388.7,Z 553.384,A -85,B 0,C 180,E1 -11608.964,E2 -11608.964} C_VEL
LIN {X 0,Y 388.7,Z 553.382,A -85,B 0,C 180,E1 -11611.036,E2 -11611.036} C_VEL
LIN {X 0,Y 388.61,Z 552.2,A -85,B 0,C 180,E1 -11613.11,E2 -11613.11} C_VEL
LIN {X 0,Y 388.661,Z 549.868,A -85,B 0,C 180,E1 -11615.187,E2 -11615.187} C_VEL
LIN {X 0,Y 388.825,Z 546.331,A -85,B 0,C 180,E1 -11617.269,E2 -11617.269} C_VEL
LIN {X 0,Y 389.026,Z 541.499,A -85,B 0,C 180,E1 -11619.357,E2 -11619.357} C_VEL
LIN {X 0,Y 389.586,Z 535.249,A -85,B 0,C 180,E1 -11621.445,E2 -11621.445} C_VEL
LIN {X 0,Y 390.238,Z 527.398,A -85,B 0,C 180,E1 -11623.54,E2 -11623.54} C_VEL
LIN {X 0,Y 391.262,Z 519.059,A -85,B 0,C 180,E1 -11625.363,E2 -11625.363} C_VEL
LIN {X 0,Y 392.478,Z 509.013,A -85,B 0,C 180,E1 -11627.185,E2 -11627.185} C_VEL
LIN {X 0,Y 393.82,Z 498.184,A -85,B 0,C 180,E1 -11628.819,E2 -11628.819} C_VEL
LIN {X 0,Y 395.309,Z 486.511,A -85,B 0,C 180,E1 -11630.284,E2 -11630.284} C_VEL
LIN {X 0,Y 396.958,Z 472.897,A -85,B 0,C 180,E1 -11631.689,E2 -11631.689} C_VEL
LIN {X 0,Y 398.475,Z 459.25,A -85,B 0,C 180,E1 -11632.831,E2 -11632.831} C_VEL
LIN {X 0,Y 399.904,Z 445.118,A -85,B 0,C 180,E1 -11633.772,E2 -11633.772} C_VEL
LIN {X 0,Y 401.133,Z 429.557,A -85,B 0,C 180,E1 -11634.567,E2 -11634.567} C_VEL
LIN {X 0,Y 402.047,Z 414.627,A -85,B 0,C 180,E1 -11635.115,E2 -11635.115} C_VEL
LIN {X 0,Y 402.654,Z 398.651,A -85,B 0,C 180,E1 -11635.489,E2 -11635.489} C_VEL
LIN {X 0,Y 405.109,Z 279.642,A -85,B 0,C 180,E1 -11637.63,E2 -11637.63} C_VEL
LIN {X 0,Y 400.712,Z 255.511,A -85,B 0,C 180,E1 -11638.437,E2 -11638.437} C_VEL
LIN {X 0,Y 398.131,Z 243.988,A -85,B 0,C 180,E1 -11638.868,E2 -11638.868} C_VEL
LIN {X 0,Y 396.891,Z 240.701,A -85,B 0,C 180,E1 -11639.07,E2 -11639.07} C_VEL
LIN {X 0,Y 393.794,Z 227.763,A -85,B 0,C 180,E1 -11641.767,E2 -11641.767} C_VEL
LIN {X 0,Y 390.072,Z 213.516,A -85,B 0,C 180,E1 -11644.912,E2 -11644.912} C_VEL
LIN {X 0,Y 390.043,Z 213.526,A -85,B 0,C 180,E1 -11647.779,E2 -11647.779} C_VEL
LIN {X 0,Y 390.073,Z 213.52,A -85,B 0,C 180,E1 -11650.824,E2 -11650.824} C_VEL
LIN {X 0,Y 390.051,Z 213.525,A -85,B 0,C 180,E1 -11653.886,E2 -11653.886} C_VEL
LIN {X 0,Y 390.075,Z 213.517,A -85,B 0,C 180,E1 -11657.619,E2 -11657.619} C_VEL
LIN {X 0,Y 390.089,Z 213.514,A -85,B 0,C 180,E1 -11660.908,E2 -11660.908} C_VEL
LIN {X 0,Y 390.079,Z 213.512,A -85,B 0,C 180,E1 -11664.793,E2 -11664.793} C_VEL
LIN {X 0,Y 390.04,Z 213.521,A -85,B 0,C 180,E1 -11668.497,E2 -11668.497} C_VEL
LIN {X 0,Y 390.11,Z 213.514,A -85,B 0,C 180,E1 -11672.07,E2 -11672.07} C_VEL
LIN {X 0,Y 390.071,Z 213.523,A -85,B 0,C 180,E1 -11675.519,E2 -11675.519} C_VEL
LIN {X 0,Y 390.079,Z 213.505,A -85,B 0,C 180,E1 -11679.53,E2 -11679.53} C_VEL
LIN {X 0,Y 390.13,Z 213.512,A -85,B 0,C 180,E1 -11683.248,E2 -11683.248} C_VEL
LIN {X 0,Y 390.186,Z 213.503,A -85,B 0,C 180,E1 -11686.561,E2 -11686.561} C_VEL
LIN {X 0,Y 390.197,Z 213.502,A -85,B 0,C 180,E1 -11690.671,E2 -11690.671} C_VEL
LIN {X 0,Y 390.319,Z 213.49,A -85,B 0,C 180,E1 -11693.798,E2 -11693.798} C_VEL
LIN {X 0,Y 390.412,Z 213.478,A -85,B 0,C 180,E1 -11697.937,E2 -11697.937} C_VEL
LIN {X 0,Y 390.543,Z 213.455,A -85,B 0,C 180,E1 -11700,E2 -11700} C_VEL
LIN {X 0,Y 390.308,Z 213.493,A -85,B 0,C 180,E1 -11703.097,E2 -11703.097} C_VEL
LIN {X 0,Y 390.296,Z 213.49,A -85,B 0,C 180,E1 -11706.65,E2 -11706.65} C_VEL
LIN {X 0,Y 390.197,Z 213.502,A -85,B 0,C 180,E1 -11709.329,E2 -11709.329} C_VEL
LIN {X 0,Y 390.163,Z 213.504,A -85,B 0,C 180,E1 -11712.483,E2 -11712.483} C_VEL
LIN {X 0,Y 390.132,Z 213.51,A -85,B 0,C 180,E1 -11715.677,E2 -11715.677} C_VEL
LIN {X 0,Y 390.098,Z 213.519,A -85,B 0,C 180,E1 -11718.923,E2 -11718.923} C_VEL
LIN {X 0,Y 390.03,Z 213.524,A -85,B 0,C 180,E1 -11722.235,E2 -11722.235} C_VEL
LIN {X 0,Y 390.112,Z 213.492,A -85,B 0,C 180,E1 -11725.744,E2 -11725.744} C_VEL
LIN {X 0,Y 390.06,Z 213.525,A -85,B 0,C 180,E1 -11729.11,E2 -11729.11} C_VEL
LIN {X 0,Y 390.038,Z 213.527,A -85,B 0,C 180,E1 -11732.722,E2 -11732.722} C_VEL
LIN {X 0,Y 390.052,Z 213.52,A -85,B 0,C 180,E1 -11735.826,E2 -11735.826} C_VEL
LIN {X 0,Y 390.065,Z 213.517,A -85,B 0,C 180,E1 -11739.219,E2 -11739.219} C_VEL
LIN {X 0,Y 390.04,Z 213.52,A -85,B 0,C 180,E1 -11742.375,E2 -11742.375} C_VEL
LIN {X 0,Y 390.045,Z 213.523,A -85,B 0,C 180,E1 -11745.356,E2 -11745.356} C_VEL
LIN {X 0,Y 390.03,Z 213.526,A -85,B 0,C 180,E1 -11748.188,E2 -11748.188} C_VEL
LIN {X 0,Y 390.088,Z 213.513,A -85,B 0,C 180,E1 -11750.909,E2 -11750.909} C_VEL
LIN {X 0,Y 390.083,Z 213.517,A -85,B 0,C 180,E1 -11754.794,E2 -11754.794} C_VEL
LIN {X 0,Y 390.094,Z 213.711,A -85,B 0,C 180,E1 -11758.654,E2 -11758.654} C_VEL
LIN {X 0,Y 392.275,Z 222.12,A -85,B 0,C 180,E1 -11760.657,E2 -11760.657} C_VEL
LIN {X 0,Y 400.212,Z 239.299,A -85,B 0,C 180,E1 -11761.644,E2 -11761.644} C_VEL
LIN {X 0,Y 405.288,Z 251.723,A -85,B 0,C 180,E1 -11762.279,E2 -11762.279} C_VEL
LIN {X 0,Y 405.551,Z 254.448,A -85,B 0,C 180,E1 -11762.352,E2 -11762.352} C_VEL
LIN {X 0,Y 403.097,Z 372.171,A -85,B 0,C 180,E1 -11764.471,E2 -11764.471} C_VEL
LIN {X 0,Y 402.513,Z 391.388,A -85,B 0,C 180,E1 -11764.881,E2 -11764.881} C_VEL
LIN {X 0,Y 401.818,Z 406.487,A -85,B 0,C 180,E1 -11765.414,E2 -11765.414} C_VEL
LIN {X 0,Y 400.891,Z 420.371,A -85,B 0,C 180,E1 -11766.09,E2 -11766.09} C_VEL
LIN {X 0,Y 399.628,Z 434.345,A -85,B 0,C 180,E1 -11766.965,E2 -11766.965} C_VEL
LIN {X 0,Y 398.349,Z 447.264,A -85,B 0,C 180,E1 -11767.982,E2 -11767.982} C_VEL
LIN {X 0,Y 396.765,Z 460.469,A -85,B 0,C 180,E1 -11769.252,E2 -11769.252} C_VEL
LIN {X 0,Y 395.3,Z 472.889,A -85,B 0,C 180,E1 -11770.72,E2 -11770.72} C_VEL
LIN {X 0,Y 393.767,Z 484.264,A -85,B 0,C 180,E1 -11772.337,E2 -11772.337} C_VEL
LIN {X 0,Y 392.418,Z 494.772,A -85,B 0,C 180,E1 -11774.15,E2 -11774.15} C_VEL
LIN {X 0,Y 391.23,Z 503.409,A -85,B 0,C 180,E1 -11775.942,E2 -11775.942} C_VEL
LIN {X 0,Y 390.633,Z 509.805,A -85,B 0,C 180,E1 -11777.532,E2 -11777.532} C_VEL
LIN {X 0,Y 389.785,Z 516.744,A -85,B 0,C 180,E1 -11779.613,E2 -11779.613} C_VEL
LIN {X 0,Y 389.308,Z 522.192,A -85,B 0,C 180,E1 -11781.696,E2 -11781.696} C_VEL
LIN {X 0,Y 388.99,Z 526.305,A -85,B 0,C 180,E1 -11783.777,E2 -11783.777} C_VEL
LIN {X 0,Y 388.754,Z 529.196,A -85,B 0,C 180,E1 -11785.853,E2 -11785.853} C_VEL
LIN {X 0,Y 388.738,Z 530.933,A -85,B 0,C 180,E1 -11787.928,E2 -11787.928} C_VEL
LIN {X 0,Y 388.716,Z 531.263,A -85,B 0,C 180,E1 -11788.686,E2 -11788.686} C_VEL
LIN {X 0,Y 388.059,Z 531.556,A -85,B 0,C 180,E1 -11789.551,E2 -11789.551} C_VEL
LIN {X 0,Y 385.186,Z 531.626,A -85,B 0,C 180,E1 -11790.957,E2 -11790.957} C_VEL
LIN {X 0,Y 382.75,Z 531.241,A -85,B 0,C 180,E1 -11792.092,E2 -11792.092} C_VEL
LIN {X 0,Y 381.708,Z 530.655,A -85,B 0,C 180,E1 -11792.967,E2 -11792.967} C_VEL
LIN {X 0,Y 381.626,Z 530.398,A -85,B 0,C 180,E1 -11793.262,E2 -11793.262} C_VEL
LIN {X 0,Y 381.806,Z 528.238,A -85,B 0,C 180,E1 -11795.281,E2 -11795.281} C_VEL
LIN {X 0,Y 382.037,Z 524.806,A -85,B 0,C 180,E1 -11797.399,E2 -11797.399} C_VEL
LIN {X 0,Y 382.45,Z 520.106,A -85,B 0,C 180,E1 -11799.519,E2 -11799.519} C_VEL
LIN {X 0,Y 383.092,Z 514.014,A -85,B 0,C 180,E1 -11801.642,E2 -11801.642} C_VEL
LIN {X 0,Y 383.953,Z 507.389,A -85,B 0,C 180,E1 -11803.496,E2 -11803.496} C_VEL
LIN {X 0,Y 385.104,Z 498.154,A -85,B 0,C 180,E1 -11805.615,E2 -11805.615} C_VEL
LIN {X 0,Y 386.5,Z 488.289,A -85,B 0,C 180,E1 -11807.459,E2 -11807.459} C_VEL
LIN {X 0,Y 388.067,Z 476.963,A -85,B 0,C 180,E1 -11809.207,E2 -11809.207} C_VEL
LIN {X 0,Y 389.482,Z 466.124,A -85,B 0,C 180,E1 -11810.601,E2 -11810.601} C_VEL
LIN {X 0,Y 391.001,Z 454.04,A -85,B 0,C 180,E1 -11811.898,E2 -11811.898} C_VEL
LIN {X 0,Y 392.458,Z 440.907,A -85,B 0,C 180,E1 -11813.062,E2 -11813.062} C_VEL
LIN {X 0,Y 393.737,Z 428.389,A -85,B 0,C 180,E1 -11813.958,E2 -11813.958} C_VEL
LIN {X 0,Y 394.902,Z 413.529,A -85,B 0,C 180,E1 -11814.803,E2 -11814.803} C_VEL
LIN {X 0,Y 395.799,Z 398.513,A -85,B 0,C 180,E1 -11815.434,E2 -11815.434} C_VEL
LIN {X 0,Y 396.492,Z 382.369,A -85,B 0,C 180,E1 -11815.879,E2 -11815.879} C_VEL
LIN {X 0,Y 398.817,Z 276.526,A -85,B 0,C 180,E1 -11817.822,E2 -11817.822} C_VEL
LIN {X 0,Y 399.176,Z 253.577,A -85,B 0,C 180,E1 -11818.253,E2 -11818.253} C_VEL
LIN {X 0,Y 391.148,Z 235.101,A -85,B 0,C 180,E1 -11819.272,E2 -11819.272} C_VEL
LIN {X 0,Y 385.002,Z 222.091,A -85,B 0,C 180,E1 -11820.092,E2 -11820.092} C_VEL
LIN {X 0,Y 383.013,Z 214.405,A -85,B 0,C 180,E1 -11821.993,E2 -11821.993} C_VEL
LIN {X 0,Y 383.016,Z 214.402,A -85,B 0,C 180,E1 -11824.667,E2 -11824.667} C_VEL
LIN {X 0,Y 382.999,Z 214.407,A -85,B 0,C 180,E1 -11827.903,E2 -11827.903} C_VEL
LIN {X 0,Y 382.982,Z 214.408,A -85,B 0,C 180,E1 -11831.346,E2 -11831.346} C_VEL
LIN {X 0,Y 382.994,Z 214.4,A -85,B 0,C 180,E1 -11834.303,E2 -11834.303} C_VEL
LIN {X 0,Y 383.006,Z 214.39,A -85,B 0,C 180,E1 -11837.239,E2 -11837.239} C_VEL
LIN {X 0,Y 383.017,Z 214.399,A -85,B 0,C 180,E1 -11840.412,E2 -11840.412} C_VEL
LIN {X 0,Y 383.021,Z 214.394,A -85,B 0,C 180,E1 -11844.044,E2 -11844.044} C_VEL
LIN {X 0,Y 382.982,Z 214.388,A -85,B 0,C 180,E1 -11847.577,E2 -11847.577} C_VEL
LIN {X 0,Y 382.991,Z 214.395,A -85,B 0,C 180,E1 -11850.3,E2 -11850.3} C_VEL
LIN {X 0,Y 383.05,Z 214.397,A -85,B 0,C 180,E1 -11852.697,E2 -11852.697} C_VEL
LIN {X 0,Y 383.045,Z 214.397,A -85,B 0,C 180,E1 -11855.039,E2 -11855.039} C_VEL
LIN {X 0,Y 382.986,Z 214.399,A -85,B 0,C 180,E1 -11858.468,E2 -11858.468} C_VEL
LIN {X 0,Y 383.055,Z 214.388,A -85,B 0,C 180,E1 -11861.826,E2 -11861.826} C_VEL
LIN {X 0,Y 383.102,Z 214.383,A -85,B 0,C 180,E1 -11865.118,E2 -11865.118} C_VEL
LIN {X 0,Y 383.091,Z 214.39,A -85,B 0,C 180,E1 -11868.358,E2 -11868.358} C_VEL
LIN {X 0,Y 383.256,Z 214.367,A -85,B 0,C 180,E1 -11871.975,E2 -11871.975} C_VEL
LIN {X 0,Y 383.191,Z 214.372,A -85,B 0,C 180,E1 -11874.738,E2 -11874.738} C_VEL
LIN {X 0,Y 383.38,Z 214.352,A -85,B 0,C 180,E1 -11877.899,E2 -11877.899} C_VEL
LIN {X 0,Y 383.513,Z 214.329,A -85,B 0,C 180,E1 -11880,E2 -11880} C_VEL
LIN {X 0,Y 383.244,Z 214.365,A -85,B 0,C 180,E1 -11883.154,E2 -11883.154} C_VEL
LIN {X 0,Y 383.275,Z 214.369,A -85,B 0,C 180,E1 -11886.316,E2 -11886.316} C_VEL
LIN {X 0,Y 383.144,Z 214.38,A -85,B 0,C 180,E1 -11889.502,E2 -11889.502} C_VEL
LIN {X 0,Y 383.117,Z 214.381,A -85,B 0,C 180,E1 -11893.536,E2 -11893.536} C_VEL
LIN {X 0,Y 383.088,Z 214.383,A -85,B 0,C 180,E1 -11897.455,E2 -11897.455} C_VEL
LIN {X 0,Y 383.021,Z 214.397,A -85,B 0,C 180,E1 -11900.647,E2 -11900.647} C_VEL
LIN {X 0,Y 383.026,Z 214.4,A -85,B 0,C 180,E1 -11903.808,E2 -11903.808} C_VEL
LIN {X 0,Y 383.073,Z 214.389,A -85,B 0,C 180,E1 -11906.124,E2 -11906.124} C_VEL
LIN {X 0,Y 383.043,Z 214.398,A -85,B 0,C 180,E1 -11908.492,E2 -11908.492} C_VEL
LIN {X 0,Y 383.002,Z 214.397,A -85,B 0,C 180,E1 -11912.428,E2 -11912.428} C_VEL
LIN {X 0,Y 383.019,Z 214.396,A -85,B 0,C 180,E1 -11915.956,E2 -11915.956} C_VEL
LIN {X 0,Y 383.009,Z 214.388,A -85,B 0,C 180,E1 -11919.587,E2 -11919.587} C_VEL
LIN {X 0,Y 383,Z 214.402,A -85,B 0,C 180,E1 -11922.779,E2 -11922.779} C_VEL
LIN {X 0,Y 382.993,Z 214.404,A -85,B 0,C 180,E1 -11925.79,E2 -11925.79} C_VEL
LIN {X 0,Y 383.011,Z 214.399,A -85,B 0,C 180,E1 -11928.792,E2 -11928.792} C_VEL
LIN {X 0,Y 382.999,Z 214.392,A -85,B 0,C 180,E1 -11932.096,E2 -11932.096} C_VEL
LIN {X 0,Y 383.053,Z 214.41,A -85,B 0,C 180,E1 -11934.574,E2 -11934.574} C_VEL
LIN {X 0,Y 386.933,Z 229.191,A -85,B 0,C 180,E1 -11937.909,E2 -11937.909} C_VEL
LIN {X 0,Y 389.63,Z 240.679,A -85,B 0,C 180,E1 -11940.36,E2 -11940.36} C_VEL
LIN {X 0,Y 392.726,Z 248.529,A -85,B 0,C 180,E1 -11940.78,E2 -11940.78} C_VEL
LIN {X 0,Y 398.434,Z 277.647,A -85,B 0,C 180,E1 -11941.819,E2 -11941.819} C_VEL
LIN {X 0,Y 398.825,Z 281.368,A -85,B 0,C 180,E1 -11941.923,E2 -11941.923} C_VEL
LIN {X 0,Y 396.063,Z 405.142,A -85,B 0,C 180,E1 -11944.196,E2 -11944.196} C_VEL
LIN {X 0,Y 395.364,Z 420.309,A -85,B 0,C 180,E1 -11944.641,E2 -11944.641} C_VEL
LIN {X 0,Y 394.364,Z 433.182,A -85,B 0,C 180,E1 -11945.172,E2 -11945.172} C_VEL
LIN {X 0,Y 393.103,Z 448.09,A -85,B 0,C 180,E1 -11946.001,E2 -11946.001} C_VEL
LIN {X 0,Y 391.543,Z 462.393,A -85,B 0,C 180,E1 -11947.021,E2 -11947.021} C_VEL
LIN {X 0,Y 390.01,Z 475.42,A -85,B 0,C 180,E1 -11948.182,E2 -11948.182} C_VEL
LIN {X 0,Y 388.447,Z 487.453,A -85,B 0,C 180,E1 -11949.48,E2 -11949.48} C_VEL
LIN {X 0,Y 386.972,Z 498.602,A -85,B 0,C 180,E1 -11950.919,E2 -11950.919} C_VEL
LIN {X 0,Y 385.633,Z 508.866,A -85,B 0,C 180,E1 -11952.5,E2 -11952.5} C_VEL
LIN {X 0,Y 384.348,Z 518.901,A -85,B 0,C 180,E1 -11954.353,E2 -11954.353} C_VEL
LIN {X 0,Y 383.187,Z 528.131,A -85,B 0,C 180,E1 -11956.426,E2 -11956.426} C_VEL
LIN {X 0,Y 382.57,Z 535.078,A -85,B 0,C 180,E1 -11958.342,E2 -11958.342} C_VEL
LIN {X 0,Y 381.97,Z 541.315,A -85,B 0,C 180,E1 -11960.468,E2 -11960.468} C_VEL
LIN {X 0,Y 381.73,Z 546.144,A -85,B 0,C 180,E1 -11962.596,E2 -11962.596} C_VEL
LIN {X 0,Y 381.571,Z 549.682,A -85,B 0,C 180,E1 -11964.716,E2 -11964.716} C_VEL
LIN {X 0,Y 381.521,Z 552.009,A -85,B 0,C 180,E1 -11966.832,E2 -11966.832} C_VEL
LIN {X 0,Y 381.614,Z 553.183,A -85,B 0,C 180,E1 -11968.945,E2 -11968.945} C_VEL
LIN {X 0,Y 381.614,Z 553.181,A -85,B 0,C 180,E1 -11971.055,E2 -11971.055} C_VEL
LIN {X 0,Y 381.521,Z 551.999,A -85,B 0,C 180,E1 -11973.168,E2 -11973.168} C_VEL
LIN {X 0,Y 381.572,Z 549.666,A -85,B 0,C 180,E1 -11975.284,E2 -11975.284} C_VEL
LIN {X 0,Y 381.731,Z 546.128,A -85,B 0,C 180,E1 -11977.404,E2 -11977.404} C_VEL
LIN {X 0,Y 381.97,Z 541.296,A -85,B 0,C 180,E1 -11979.532,E2 -11979.532} C_VEL
LIN {X 0,Y 382.567,Z 535.045,A -85,B 0,C 180,E1 -11981.658,E2 -11981.658} C_VEL
LIN {X 0,Y 383.273,Z 527.194,A -85,B 0,C 180,E1 -11983.791,E2 -11983.791} C_VEL
LIN {X 0,Y 384.35,Z 518.854,A -85,B 0,C 180,E1 -11985.647,E2 -11985.647} C_VEL
LIN {X 0,Y 385.65,Z 508.809,A -85,B 0,C 180,E1 -11987.499,E2 -11987.499} C_VEL
LIN {X 0,Y 386.972,Z 498.538,A -85,B 0,C 180,E1 -11989.081,E2 -11989.081} C_VEL
LIN {X 0,Y 388.606,Z 486.306,A -85,B 0,C 180,E1 -11990.65,E2 -11990.65} C_VEL
LIN {X 0,Y 390.331,Z 472.691,A -85,B 0,C 180,E1 -11992.077,E2 -11992.077} C_VEL
LIN {X 0,Y 391.902,Z 459.043,A -85,B 0,C 180,E1 -11993.236,E2 -11993.236} C_VEL
LIN {X 0,Y 393.415,Z 444.911,A -85,B 0,C 180,E1 -11994.189,E2 -11994.189} C_VEL
LIN {X 0,Y 394.67,Z 429.479,A -85,B 0,C 180,E1 -11994.991,E2 -11994.991} C_VEL
LIN {X 0,Y 395.618,Z 414.413,A -85,B 0,C 180,E1 -11995.552,E2 -11995.552} C_VEL
LIN {X 0,Y 396.25,Z 398.43,A -85,B 0,C 180,E1 -11995.932,E2 -11995.932} C_VEL
LIN {X 0,Y 398.808,Z 280.266,A -85,B 0,C 180,E1 -11998.088,E2 -11998.088} C_VEL
LIN {X 0,Y 394.126,Z 255.253,A -85,B 0,C 180,E1 -11998.957,E2 -11998.957} C_VEL
LIN {X 0,Y 392.175,Z 246.715,A -85,B 0,C 180,E1 -11999.288,E2 -11999.288} C_VEL
LIN {X 0,Y 389.634,Z 240.628,A -85,B 0,C 180,E1 -11999.635,E2 -11999.635} C_VEL
LIN {X 0,Y 386.091,Z 225.922,A -85,B 0,C 180,E1 -12002.794,E2 -12002.794} C_VEL
LIN {X 0,Y 383.03,Z 214.394,A -85,B 0,C 180,E1 -12005.468,E2 -12005.468} C_VEL
LIN {X 0,Y 383.005,Z 214.403,A -85,B 0,C 180,E1 -12008.6,E2 -12008.6} C_VEL
LIN {X 0,Y 383.009,Z 214.399,A -85,B 0,C 180,E1 -12011.343,E2 -12011.343} C_VEL
LIN {X 0,Y 382.991,Z 214.402,A -85,B 0,C 180,E1 -12014.303,E2 -12014.303} C_VEL
LIN {X 0,Y 383.034,Z 214.392,A -85,B 0,C 180,E1 -12017.244,E2 -12017.244} C_VEL
LIN {X 0,Y 383.016,Z 214.396,A -85,B 0,C 180,E1 -12020.412,E2 -12020.412} C_VEL
LIN {X 0,Y 383.02,Z 214.393,A -85,B 0,C 180,E1 -12024.044,E2 -12024.044} C_VEL
LIN {X 0,Y 383.03,Z 214.394,A -85,B 0,C 180,E1 -12027.852,E2 -12027.852} C_VEL
LIN {X 0,Y 383.057,Z 214.396,A -85,B 0,C 180,E1 -12031.72,E2 -12031.72} C_VEL
LIN {X 0,Y 383.044,Z 214.395,A -85,B 0,C 180,E1 -12035.039,E2 -12035.039} C_VEL
LIN {X 0,Y 382.984,Z 214.381,A -85,B 0,C 180,E1 -12038.469,E2 -12038.469} C_VEL
LIN {X 0,Y 383.081,Z 214.393,A -85,B 0,C 180,E1 -12041.827,E2 -12041.827} C_VEL
LIN {X 0,Y 383.102,Z 214.387,A -85,B 0,C 180,E1 -12045.118,E2 -12045.118} C_VEL
LIN {X 0,Y 383.09,Z 214.387,A -85,B 0,C 180,E1 -12048.358,E2 -12048.358} C_VEL
LIN {X 0,Y 383.256,Z 214.366,A -85,B 0,C 180,E1 -12051.975,E2 -12051.975} C_VEL
LIN {X 0,Y 383.191,Z 214.376,A -85,B 0,C 180,E1 -12054.738,E2 -12054.738} C_VEL
LIN {X 0,Y 383.38,Z 214.354,A -85,B 0,C 180,E1 -12057.899,E2 -12057.899} C_VEL
LIN {X 0,Y 383.513,Z 214.331,A -85,B 0,C 180,E1 -12060,E2 -12060} C_VEL
LIN {X 0,Y 383.244,Z 214.372,A -85,B 0,C 180,E1 -12063.154,E2 -12063.154} C_VEL
LIN {X 0,Y 383.255,Z 214.366,A -85,B 0,C 180,E1 -12066.642,E2 -12066.642} C_VEL
LIN {X 0,Y 383.144,Z 214.382,A -85,B 0,C 180,E1 -12069.502,E2 -12069.502} C_VEL
LIN {X 0,Y 383.118,Z 214.386,A -85,B 0,C 180,E1 -12073.536,E2 -12073.536} C_VEL
LIN {X 0,Y 383.087,Z 214.389,A -85,B 0,C 180,E1 -12077.455,E2 -12077.455} C_VEL
LIN {X 0,Y 383.021,Z 214.395,A -85,B 0,C 180,E1 -12080.647,E2 -12080.647} C_VEL
LIN {X 0,Y 383.019,Z 214.394,A -85,B 0,C 180,E1 -12083.808,E2 -12083.808} C_VEL
LIN {X 0,Y 383.073,Z 214.367,A -85,B 0,C 180,E1 -12086.124,E2 -12086.124} C_VEL
LIN {X 0,Y 383.044,Z 214.392,A -85,B 0,C 180,E1 -12088.493,E2 -12088.493} C_VEL
LIN {X 0,Y 383.005,Z 214.399,A -85,B 0,C 180,E1 -12092.15,E2 -12092.15} C_VEL
LIN {X 0,Y 383.013,Z 214.397,A -85,B 0,C 180,E1 -12094.669,E2 -12094.669} C_VEL
LIN {X 0,Y 382.996,Z 214.398,A -85,B 0,C 180,E1 -12097.905,E2 -12097.905} C_VEL
LIN {X 0,Y 382.98,Z 214.399,A -85,B 0,C 180,E1 -12101.348,E2 -12101.348} C_VEL
LIN {X 0,Y 382.996,Z 214.399,A -85,B 0,C 180,E1 -12104.305,E2 -12104.305} C_VEL
LIN {X 0,Y 383.007,Z 214.402,A -85,B 0,C 180,E1 -12107.241,E2 -12107.241} C_VEL
LIN {X 0,Y 383.013,Z 214.396,A -85,B 0,C 180,E1 -12110.414,E2 -12110.414} C_VEL
LIN {X 0,Y 383.023,Z 214.394,A -85,B 0,C 180,E1 -12114.045,E2 -12114.045} C_VEL
LIN {X 0,Y 382.985,Z 214.405,A -85,B 0,C 180,E1 -12117.579,E2 -12117.579} C_VEL
LIN {X 0,Y 383.018,Z 214.618,A -85,B 0,C 180,E1 -12118.162,E2 -12118.162} C_VEL
LIN {X 0,Y 385.118,Z 222.438,A -85,B 0,C 180,E1 -12120.058,E2 -12120.058} C_VEL
LIN {X 0,Y 393.889,Z 241.092,A -85,B 0,C 180,E1 -12121.179,E2 -12121.179} C_VEL
LIN {X 0,Y 399.214,Z 253.924,A -85,B 0,C 180,E1 -12121.859,E2 -12121.859} C_VEL
LIN {X 0,Y 397.574,Z 333.093,A -85,B 0,C 180,E1 -12123.314,E2 -12123.314} C_VEL
LIN {X 0,Y 396.316,Z 387.011,A -85,B 0,C 180,E1 -12124.32,E2 -12124.32} C_VEL
LIN {X 0,Y 395.587,Z 402.921,A -85,B 0,C 180,E1 -12124.826,E2 -12124.826} C_VEL
LIN {X 0,Y 394.649,Z 417.131,A -85,B 0,C 180,E1 -12125.476,E2 -12125.476} C_VEL
LIN {X 0,Y 393.487,Z 430.908,A -85,B 0,C 180,E1 -12126.306,E2 -12126.306} C_VEL
LIN {X 0,Y 392.111,Z 444.483,A -85,B 0,C 180,E1 -12127.335,E2 -12127.335} C_VEL
LIN {X 0,Y 390.62,Z 456.967,A -85,B 0,C 180,E1 -12128.495,E2 -12128.495} C_VEL
LIN {X 0,Y 389.108,Z 468.547,A -85,B 0,C 180,E1 -12129.792,E2 -12129.792} C_VEL
LIN {X 0,Y 387.7,Z 479.296,A -85,B 0,C 180,E1 -12131.231,E2 -12131.231} C_VEL
LIN {X 0,Y 386.336,Z 489.232,A -85,B 0,C 180,E1 -12132.806,E2 -12132.806} C_VEL
LIN {X 0,Y 385.007,Z 498.931,A -85,B 0,C 180,E1 -12134.652,E2 -12134.652} C_VEL
LIN {X 0,Y 383.959,Z 507.012,A -85,B 0,C 180,E1 -12136.504,E2 -12136.504} C_VEL
LIN {X 0,Y 383.106,Z 513.678,A -85,B 0,C 180,E1 -12138.358,E2 -12138.358} C_VEL
LIN {X 0,Y 382.457,Z 519.847,A -85,B 0,C 180,E1 -12140.481,E2 -12140.481} C_VEL
LIN {X 0,Y 382.057,Z 524.61,A -85,B 0,C 180,E1 -12142.602,E2 -12142.602} C_VEL
LIN {X 0,Y 381.815,Z 528.099,A -85,B 0,C 180,E1 -12144.719,E2 -12144.719} C_VEL
LIN {X 0,Y 381.627,Z 530.408,A -85,B 0,C 180,E1 -12146.833,E2 -12146.833} C_VEL
LIN {X 0,Y 381.64,Z 531.584,A -85,B 0,C 180,E1 -12148.945,E2 -12148.945} C_VEL
LIN {X 0,Y 381.641,Z 531.6,A -85,B 0,C 180,E1 -12151.055,E2 -12151.055} C_VEL
LIN {X 0,Y 381.626,Z 530.398,A -85,B 0,C 180,E1 -12153.262,E2 -12153.262} C_VEL
LIN {X 0,Y 380.983,Z 529.638,A -85,B 0,C 180,E1 -12154.135,E2 -12154.135} C_VEL
LIN {X 0,Y 378.226,Z 528.04,A -85,B 0,C 180,E1 -12155.554,E2 -12155.554} C_VEL
LIN {X 0,Y 375.951,Z 526.439,A -85,B 0,C 180,E1 -12156.69,E2 -12156.69} C_VEL
LIN {X 0,Y 375.056,Z 524.973,A -85,B 0,C 180,E1 -12157.558,E2 -12157.558} C_VEL
LIN {X 0,Y 375.027,Z 524.401,A -85,B 0,C 180,E1 -12157.848,E2 -12157.848} C_VEL
LIN {X 0,Y 375.424,Z 520.306,A -85,B 0,C 180,E1 -12159.699,E2 -12159.699} C_VEL
LIN {X 0,Y 376.122,Z 514.213,A -85,B 0,C 180,E1 -12161.861,E2 -12161.861} C_VEL
LIN {X 0,Y 376.977,Z 507.59,A -85,B 0,C 180,E1 -12163.75,E2 -12163.75} C_VEL
LIN {X 0,Y 378.05,Z 499.584,A -85,B 0,C 180,E1 -12165.638,E2 -12165.638} C_VEL
LIN {X 0,Y 379.484,Z 489.973,A -85,B 0,C 180,E1 -12167.514,E2 -12167.514} C_VEL
LIN {X 0,Y 380.898,Z 480.143,A -85,B 0,C 180,E1 -12169.117,E2 -12169.117} C_VEL
LIN {X 0,Y 382.39,Z 469.514,A -85,B 0,C 180,E1 -12170.579,E2 -12170.579} C_VEL
LIN {X 0,Y 384.102,Z 456.806,A -85,B 0,C 180,E1 -12172.029,E2 -12172.029} C_VEL
LIN {X 0,Y 385.596,Z 444.253,A -85,B 0,C 180,E1 -12173.212,E2 -12173.212} C_VEL
LIN {X 0,Y 387.059,Z 430.565,A -85,B 0,C 180,E1 -12174.255,E2 -12174.255} C_VEL
LIN {X 0,Y 388.287,Z 416.542,A -85,B 0,C 180,E1 -12175.1,E2 -12175.1} C_VEL
LIN {X 0,Y 389.216,Z 402.349,A -85,B 0,C 180,E1 -12175.752,E2 -12175.752} C_VEL
LIN {X 0,Y 390.014,Z 387.036,A -85,B 0,C 180,E1 -12176.234,E2 -12176.234} C_VEL
LIN {X 0,Y 392.5,Z 279.402,A -85,B 0,C 180,E1 -12178.254,E2 -12178.254} C_VEL
LIN {X 0,Y 392.979,Z 255.72,A -85,B 0,C 180,E1 -12178.699,E2 -12178.699} C_VEL
LIN {X 0,Y 385.658,Z 238.746,A -85,B 0,C 180,E1 -12179.657,E2 -12179.657} C_VEL
LIN {X 0,Y 377.811,Z 222.367,A -85,B 0,C 180,E1 -12180.714,E2 -12180.714} C_VEL
LIN {X 0,Y 375.948,Z 215.284,A -85,B 0,C 180,E1 -12182.57,E2 -12182.57} C_VEL
LIN {X 0,Y 375.956,Z 215.287,A -85,B 0,C 180,E1 -12185.415,E2 -12185.415} C_VEL
LIN {X 0,Y 375.973,Z 215.281,A -85,B 0,C 180,E1 -12188.27,E2 -12188.27} C_VEL
LIN {X 0,Y 375.932,Z 215.285,A -85,B 0,C 180,E1 -12191.6,E2 -12191.6} C_VEL
LIN {X 0,Y 375.95,Z 215.282,A -85,B 0,C 180,E1 -12195.264,E2 -12195.264} C_VEL
LIN {X 0,Y 375.971,Z 215.274,A -85,B 0,C 180,E1 -12199.137,E2 -12199.137} C_VEL
LIN {X 0,Y 375.963,Z 215.264,A -85,B 0,C 180,E1 -12201.911,E2 -12201.911} C_VEL
LIN {X 0,Y 375.975,Z 215.279,A -85,B 0,C 180,E1 -12205.332,E2 -12205.332} C_VEL
LIN {X 0,Y 375.954,Z 215.258,A -85,B 0,C 180,E1 -12208.438,E2 -12208.438} C_VEL
LIN {X 0,Y 375.996,Z 215.273,A -85,B 0,C 180,E1 -12212.141,E2 -12212.141} C_VEL
LIN {X 0,Y 375.999,Z 215.269,A -85,B 0,C 180,E1 -12214.538,E2 -12214.538} C_VEL
LIN {X 0,Y 375.956,Z 215.273,A -85,B 0,C 180,E1 -12218.045,E2 -12218.045} C_VEL
LIN {X 0,Y 376.001,Z 215.267,A -85,B 0,C 180,E1 -12221.473,E2 -12221.473} C_VEL
LIN {X 0,Y 376.051,Z 215.264,A -85,B 0,C 180,E1 -12224.832,E2 -12224.832} C_VEL
LIN {X 0,Y 376.043,Z 215.267,A -85,B 0,C 180,E1 -12228.136,E2 -12228.136} C_VEL
LIN {X 0,Y 376.212,Z 215.245,A -85,B 0,C 180,E1 -12231.918,E2 -12231.918} C_VEL
LIN {X 0,Y 376.163,Z 215.247,A -85,B 0,C 180,E1 -12234.64,E2 -12234.64} C_VEL
LIN {X 0,Y 376.346,Z 215.228,A -85,B 0,C 180,E1 -12237.859,E2 -12237.859} C_VEL
LIN {X 0,Y 376.482,Z 215.205,A -85,B 0,C 180,E1 -12240,E2 -12240} C_VEL
LIN {X 0,Y 376.182,Z 215.244,A -85,B 0,C 180,E1 -12243.213,E2 -12243.213} C_VEL
LIN {X 0,Y 376.233,Z 215.247,A -85,B 0,C 180,E1 -12246.435,E2 -12246.435} C_VEL
LIN {X 0,Y 376.111,Z 215.256,A -85,B 0,C 180,E1 -12249.682,E2 -12249.682} C_VEL
LIN {X 0,Y 376.081,Z 215.258,A -85,B 0,C 180,E1 -12253.658,E2 -12253.658} C_VEL
LIN {X 0,Y 376.037,Z 215.261,A -85,B 0,C 180,E1 -12257.608,E2 -12257.608} C_VEL
LIN {X 0,Y 375.971,Z 215.273,A -85,B 0,C 180,E1 -12260.832,E2 -12260.832} C_VEL
LIN {X 0,Y 375.986,Z 215.277,A -85,B 0,C 180,E1 -12264.282,E2 -12264.282} C_VEL
LIN {X 0,Y 376.013,Z 215.274,A -85,B 0,C 180,E1 -12266.653,E2 -12266.653} C_VEL
LIN {X 0,Y 375.97,Z 215.277,A -85,B 0,C 180,E1 -12269.079,E2 -12269.079} C_VEL
LIN {X 0,Y 375.95,Z 215.273,A -85,B 0,C 180,E1 -12272.828,E2 -12272.828} C_VEL
LIN {X 0,Y 375.951,Z 215.278,A -85,B 0,C 180,E1 -12275.416,E2 -12275.416} C_VEL
LIN {X 0,Y 375.968,Z 215.276,A -85,B 0,C 180,E1 -12278.271,E2 -12278.271} C_VEL
LIN {X 0,Y 375.928,Z 215.27,A -85,B 0,C 180,E1 -12281.601,E2 -12281.601} C_VEL
LIN {X 0,Y 375.922,Z 215.283,A -85,B 0,C 180,E1 -12285.269,E2 -12285.269} C_VEL
LIN {X 0,Y 375.956,Z 215.277,A -85,B 0,C 180,E1 -12288.395,E2 -12288.395} C_VEL
LIN {X 0,Y 375.974,Z 215.27,A -85,B 0,C 180,E1 -12291.729,E2 -12291.729} C_VEL
LIN {X 0,Y 376.018,Z 215.374,A -85,B 0,C 180,E1 -12294.056,E2 -12294.056} C_VEL
LIN {X 0,Y 379.702,Z 229.343,A -85,B 0,C 180,E1 -12297.298,E2 -12297.298} C_VEL
LIN {X 0,Y 382.397,Z 240.485,A -85,B 0,C 180,E1 -12299.746,E2 -12299.746} C_VEL
LIN {X 0,Y 386.763,Z 250.915,A -85,B 0,C 180,E1 -12300.338,E2 -12300.338} C_VEL
LIN {X 0,Y 392.524,Z 280.706,A -85,B 0,C 180,E1 -12301.421,E2 -12301.421} C_VEL
LIN {X 0,Y 389.94,Z 397.046,A -85,B 0,C 180,E1 -12303.581,E2 -12303.581} C_VEL
LIN {X 0,Y 389.391,Z 412.301,A -85,B 0,C 180,E1 -12303.937,E2 -12303.937} C_VEL
LIN {X 0,Y 388.331,Z 427.833,A -85,B 0,C 180,E1 -12304.494,E2 -12304.494} C_VEL
LIN {X 0,Y 387.101,Z 442.76,A -85,B 0,C 180,E1 -12305.255,E2 -12305.255} C_VEL
LIN {X 0,Y 385.588,Z 457.276,A -85,B 0,C 180,E1 -12306.222,E2 -12306.222} C_VEL
LIN {X 0,Y 383.902,Z 471.168,A -85,B 0,C 180,E1 -12307.391,E2 -12307.391} C_VEL
LIN {X 0,Y 382.28,Z 483.857,A -85,B 0,C 180,E1 -12308.71,E2 -12308.71} C_VEL
LIN {X 0,Y 380.76,Z 494.533,A -85,B 0,C 180,E1 -12310.035,E2 -12310.035} C_VEL
LIN {X 0,Y 379.301,Z 505.395,A -85,B 0,C 180,E1 -12311.64,E2 -12311.64} C_VEL
LIN {X 0,Y 377.955,Z 514.613,A -85,B 0,C 180,E1 -12313.249,E2 -12313.249} C_VEL
LIN {X 0,Y 376.769,Z 523.661,A -85,B 0,C 180,E1 -12315.139,E2 -12315.139} C_VEL
LIN {X 0,Y 375.913,Z 531.172,A -85,B 0,C 180,E1 -12317.036,E2 -12317.036} C_VEL
LIN {X 0,Y 375.155,Z 538.18,A -85,B 0,C 180,E1 -12319.203,E2 -12319.203} C_VEL
LIN {X 0,Y 374.756,Z 543.695,A -85,B 0,C 180,E1 -12321.372,E2 -12321.372} C_VEL
LIN {X 0,Y 374.563,Z 547.868,A -85,B 0,C 180,E1 -12323.536,E2 -12323.536} C_VEL
LIN {X 0,Y 374.478,Z 550.793,A -85,B 0,C 180,E1 -12325.695,E2 -12325.695} C_VEL
LIN {X 0,Y 374.45,Z 552.538,A -85,B 0,C 180,E1 -12327.849,E2 -12327.849} C_VEL
LIN {X 0,Y 374.551,Z 553.138,A -85,B 0,C 180,E1 -12330,E2 -12330} C_VEL
LIN {X 0,Y 374.45,Z 552.531,A -85,B 0,C 180,E1 -12332.151,E2 -12332.151} C_VEL
LIN {X 0,Y 374.479,Z 550.779,A -85,B 0,C 180,E1 -12334.305,E2 -12334.305} C_VEL
LIN {X 0,Y 374.563,Z 547.85,A -85,B 0,C 180,E1 -12336.464,E2 -12336.464} C_VEL
LIN {X 0,Y 374.756,Z 543.678,A -85,B 0,C 180,E1 -12338.628,E2 -12338.628} C_VEL
LIN {X 0,Y 375.155,Z 538.152,A -85,B 0,C 180,E1 -12340.797,E2 -12340.797} C_VEL
LIN {X 0,Y 375.896,Z 531.128,A -85,B 0,C 180,E1 -12342.965,E2 -12342.965} C_VEL
LIN {X 0,Y 376.768,Z 523.615,A -85,B 0,C 180,E1 -12344.861,E2 -12344.861} C_VEL
LIN {X 0,Y 377.958,Z 514.562,A -85,B 0,C 180,E1 -12346.751,E2 -12346.751} C_VEL
LIN {X 0,Y 379.52,Z 503.741,A -85,B 0,C 180,E1 -12348.62,E2 -12348.62} C_VEL
LIN {X 0,Y 381.133,Z 491.576,A -85,B 0,C 180,E1 -12350.354,E2 -12350.354} C_VEL
LIN {X 0,Y 382.885,Z 479.012,A -85,B 0,C 180,E1 -12351.82,E2 -12351.82} C_VEL
LIN {X 0,Y 384.459,Z 466.76,A -85,B 0,C 180,E1 -12353,E2 -12353} C_VEL
LIN {X 0,Y 385.965,Z 453.686,A -85,B 0,C 180,E1 -12354.03,E2 -12354.03} C_VEL
LIN {X 0,Y 387.376,Z 439.512,A -85,B 0,C 180,E1 -12354.92,E2 -12354.92} C_VEL
LIN {X 0,Y 388.552,Z 424.229,A -85,B 0,C 180,E1 -12355.649,E2 -12355.649} C_VEL
LIN {X 0,Y 389.471,Z 409.629,A -85,B 0,C 180,E1 -12356.129,E2 -12356.129} C_VEL
LIN {X 0,Y 390.206,Z 385.676,A -85,B 0,C 180,E1 -12356.616,E2 -12356.616} C_VEL
LIN {X 0,Y 392.569,Z 281.559,A -85,B 0,C 180,E1 -12358.545,E2 -12358.545} C_VEL
LIN {X 0,Y 387.984,Z 256.9,A -85,B 0,C 180,E1 -12359.421,E2 -12359.421} C_VEL
LIN {X 0,Y 386.19,Z 249.208,A -85,B 0,C 180,E1 -12359.731,E2 -12359.731} C_VEL
LIN {X 0,Y 382.407,Z 240.375,A -85,B 0,C 180,E1 -12360.256,E2 -12360.256} C_VEL
LIN {X 0,Y 378.882,Z 226.113,A -85,B 0,C 180,E1 -12363.414,E2 -12363.414} C_VEL
LIN {X 0,Y 375.998,Z 215.273,A -85,B 0,C 180,E1 -12365.987,E2 -12365.987} C_VEL
LIN {X 0,Y 375.965,Z 215.278,A -85,B 0,C 180,E1 -12369.461,E2 -12369.461} C_VEL
LIN {X 0,Y 375.957,Z 215.28,A -85,B 0,C 180,E1 -12372.296,E2 -12372.296} C_VEL
LIN {X 0,Y 375.934,Z 215.281,A -85,B 0,C 180,E1 -12376.235,E2 -12376.235} C_VEL
LIN {X 0,Y 375.992,Z 215.272,A -85,B 0,C 180,E1 -12380.027,E2 -12380.027} C_VEL
LIN {X 0,Y 375.959,Z 215.276,A -85,B 0,C 180,E1 -12383.495,E2 -12383.495} C_VEL
LIN {X 0,Y 375.958,Z 215.277,A -85,B 0,C 180,E1 -12385.888,E2 -12385.888} C_VEL
LIN {X 0,Y 375.963,Z 215.274,A -85,B 0,C 180,E1 -12389.687,E2 -12389.687} C_VEL
LIN {X 0,Y 375.995,Z 215.271,A -85,B 0,C 180,E1 -12392.141,E2 -12392.141} C_VEL
LIN {X 0,Y 375.998,Z 215.272,A -85,B 0,C 180,E1 -12394.539,E2 -12394.539} C_VEL
LIN {X 0,Y 375.95,Z 215.257,A -85,B 0,C 180,E1 -12398.045,E2 -12398.045} C_VEL
LIN {X 0,Y 376.016,Z 215.272,A -85,B 0,C 180,E1 -12401.474,E2 -12401.474} C_VEL
LIN {X 0,Y 376.05,Z 215.264,A -85,B 0,C 180,E1 -12404.832,E2 -12404.832} C_VEL
LIN {X 0,Y 376.042,Z 215.266,A -85,B 0,C 180,E1 -12408.136,E2 -12408.136} C_VEL
LIN {X 0,Y 376.211,Z 215.243,A -85,B 0,C 180,E1 -12411.919,E2 -12411.919} C_VEL
LIN {X 0,Y 376.163,Z 215.251,A -85,B 0,C 180,E1 -12414.64,E2 -12414.64} C_VEL
LIN {X 0,Y 376.346,Z 215.23,A -85,B 0,C 180,E1 -12417.86,E2 -12417.86} C_VEL
LIN {X 0,Y 376.482,Z 215.206,A -85,B 0,C 180,E1 -12420,E2 -12420} C_VEL
LIN {X 0,Y 376.182,Z 215.25,A -85,B 0,C 180,E1 -12423.213,E2 -12423.213} C_VEL
LIN {X 0,Y 376.22,Z 215.243,A -85,B 0,C 180,E1 -12426.631,E2 -12426.631} C_VEL
LIN {X 0,Y 376.112,Z 215.26,A -85,B 0,C 180,E1 -12429.682,E2 -12429.682} C_VEL
LIN {X 0,Y 376.082,Z 215.263,A -85,B 0,C 180,E1 -12433.658,E2 -12433.658} C_VEL
LIN {X 0,Y 376.036,Z 215.268,A -85,B 0,C 180,E1 -12437.607,E2 -12437.607} C_VEL
LIN {X 0,Y 375.971,Z 215.273,A -85,B 0,C 180,E1 -12440.833,E2 -12440.833} C_VEL
LIN {X 0,Y 375.983,Z 215.27,A -85,B 0,C 180,E1 -12444.282,E2 -12444.282} C_VEL
LIN {X 0,Y 376.013,Z 215.249,A -85,B 0,C 180,E1 -12446.653,E2 -12446.653} C_VEL
LIN {X 0,Y 375.971,Z 215.28,A -85,B 0,C 180,E1 -12449.079,E2 -12449.079} C_VEL
LIN {X 0,Y 375.944,Z 215.283,A -85,B 0,C 180,E1 -12452.829,E2 -12452.829} C_VEL
LIN {X 0,Y 375.953,Z 215.278,A -85,B 0,C 180,E1 -12455.416,E2 -12455.416} C_VEL
LIN {X 0,Y 375.97,Z 215.275,A -85,B 0,C 180,E1 -12458.271,E2 -12458.271} C_VEL
LIN {X 0,Y 375.93,Z 215.276,A -85,B 0,C 180,E1 -12461.601,E2 -12461.601} C_VEL
LIN {X 0,Y 375.952,Z 215.279,A -85,B 0,C 180,E1 -12465.265,E2 -12465.265} C_VEL
LIN {X 0,Y 375.938,Z 215.284,A -85,B 0,C 180,E1 -12469.134,E2 -12469.134} C_VEL
LIN {X 0,Y 375.962,Z 215.277,A -85,B 0,C 180,E1 -12471.912,E2 -12471.912} C_VEL
LIN {X 0,Y 375.978,Z 215.279,A -85,B 0,C 180,E1 -12475.333,E2 -12475.333} C_VEL
LIN {X 0,Y 375.95,Z 215.339,A -85,B 0,C 180,E1 -12477.607,E2 -12477.607} C_VEL
LIN {X 0,Y 377.855,Z 222.491,A -85,B 0,C 180,E1 -12479.417,E2 -12479.417} C_VEL
LIN {X 0,Y 387.693,Z 243.15,A -85,B 0,C 180,E1 -12480.712,E2 -12480.712} C_VEL
LIN {X 0,Y 392.943,Z 255.64,A -85,B 0,C 180,E1 -12481.4,E2 -12481.4} C_VEL
LIN {X 0,Y 391.249,Z 333.319,A -85,B 0,C 180,E1 -12482.847,E2 -12482.847} C_VEL
LIN {X 0,Y 389.945,Z 387.23,A -85,B 0,C 180,E1 -12483.869,E2 -12483.869} C_VEL
LIN {X 0,Y 389.196,Z 402.734,A -85,B 0,C 180,E1 -12484.365,E2 -12484.365} C_VEL
LIN {X 0,Y 388.156,Z 417.98,A -85,B 0,C 180,E1 -12485.075,E2 -12485.075} C_VEL
LIN {X 0,Y 386.821,Z 432.998,A -85,B 0,C 180,E1 -12486.014,E2 -12486.014} C_VEL
LIN {X 0,Y 385.407,Z 446.247,A -85,B 0,C 180,E1 -12487.06,E2 -12487.06} C_VEL
LIN {X 0,Y 383.657,Z 459.711,A -85,B 0,C 180,E1 -12488.368,E2 -12488.368} C_VEL
LIN {X 0,Y 382.125,Z 471.098,A -85,B 0,C 180,E1 -12489.717,E2 -12489.717} C_VEL
LIN {X 0,Y 380.698,Z 481.273,A -85,B 0,C 180,E1 -12491.152,E2 -12491.152} C_VEL
LIN {X 0,Y 379.316,Z 490.912,A -85,B 0,C 180,E1 -12492.756,E2 -12492.756} C_VEL
LIN {X 0,Y 377.939,Z 500.357,A -85,B 0,C 180,E1 -12494.634,E2 -12494.634} C_VEL
LIN {X 0,Y 376.915,Z 508.216,A -85,B 0,C 180,E1 -12496.522,E2 -12496.522} C_VEL
LIN {X 0,Y 375.914,Z 515.553,A -85,B 0,C 180,E1 -12498.679,E2 -12498.679} C_VEL
LIN {X 0,Y 375.313,Z 521.369,A -85,B 0,C 180,E1 -12500.842,E2 -12500.842} C_VEL
LIN {X 0,Y 374.993,Z 524.812,A -85,B 0,C 180,E1 -12502.462,E2 -12502.462} C_VEL
LIN {X 0,Y 374.743,Z 528.3,A -85,B 0,C 180,E1 -12504.62,E2 -12504.62} C_VEL
LIN {X 0,Y 374.538,Z 530.609,A -85,B 0,C 180,E1 -12506.773,E2 -12506.773} C_VEL
LIN {X 0,Y 374.542,Z 531.785,A -85,B 0,C 180,E1 -12508.925,E2 -12508.925} C_VEL
LIN {X 0,Y 374.543,Z 531.801,A -85,B 0,C 180,E1 -12511.075,E2 -12511.075} C_VEL
LIN {X 0,Y 374.537,Z 530.648,A -85,B 0,C 180,E1 -12513.269,E2 -12513.269} C_VEL
LIN {X 0,Y 374.731,Z 528.438,A -85,B 0,C 180,E1 -12515.381,E2 -12515.381} C_VEL
LIN {X 0,Y 374.975,Z 525.006,A -85,B 0,C 180,E1 -12517.539,E2 -12517.539} C_VEL
LIN {X 0,Y 375.027,Z 524.401,A -85,B 0,C 180,E1 -12517.848,E2 -12517.848} C_VEL
LIN {X 0,Y 374.521,Z 522.698,A -85,B 0,C 180,E1 -12518.71,E2 -12518.71} C_VEL
LIN {X 0,Y 371.959,Z 519.674,A -85,B 0,C 180,E1 -12520.108,E2 -12520.108} C_VEL
LIN {X 0,Y 369.551,Z 516.152,A -85,B 0,C 180,E1 -12521.495,E2 -12521.495} C_VEL
LIN {X 0,Y 369.29,Z 513.639,A -85,B 0,C 180,E1 -12522.324,E2 -12522.324} C_VEL
LIN {X 0,Y 370.141,Z 506.74,A -85,B 0,C 180,E1 -12524.29,E2 -12524.29} C_VEL
LIN {X 0,Y 371.381,Z 498.553,A -85,B 0,C 180,E1 -12526.208,E2 -12526.208} C_VEL
LIN {X 0,Y 372.923,Z 488.687,A -85,B 0,C 180,E1 -12528.116,E2 -12528.116} C_VEL
LIN {X 0,Y 374.46,Z 478.569,A -85,B 0,C 180,E1 -12529.744,E2 -12529.744} C_VEL
LIN {X 0,Y 376.036,Z 467.583,A -85,B 0,C 180,E1 -12531.229,E2 -12531.229} C_VEL
LIN {X 0,Y 377.674,Z 455.718,A -85,B 0,C 180,E1 -12532.569,E2 -12532.569} C_VEL
LIN {X 0,Y 379.251,Z 442.873,A -85,B 0,C 180,E1 -12533.769,E2 -12533.769} C_VEL
LIN {X 0,Y 380.79,Z 428.777,A -85,B 0,C 180,E1 -12534.827,E2 -12534.827} C_VEL
LIN {X 0,Y 381.994,Z 414.965,A -85,B 0,C 180,E1 -12535.642,E2 -12535.642} C_VEL
LIN {X 0,Y 382.993,Z 399.802,A -85,B 0,C 180,E1 -12536.312,E2 -12536.312} C_VEL
LIN {X 0,Y 383.737,Z 384.23,A -85,B 0,C 180,E1 -12536.77,E2 -12536.77} C_VEL
LIN {X 0,Y 386.217,Z 283.154,A -85,B 0,C 180,E1 -12538.682,E2 -12538.682} C_VEL
LIN {X 0,Y 386.669,Z 257.431,A -85,B 0,C 180,E1 -12539.181,E2 -12539.181} C_VEL
LIN {X 0,Y 380.134,Z 242.357,A -85,B 0,C 180,E1 -12540.058,E2 -12540.058} C_VEL
LIN {X 0,Y 370.618,Z 222.666,A -85,B 0,C 180,E1 -12541.361,E2 -12541.361} C_VEL
LIN {X 0,Y 368.909,Z 216.163,A -85,B 0,C 180,E1 -12543.092,E2 -12543.092} C_VEL
LIN {X 0,Y 368.916,Z 216.155,A -85,B 0,C 180,E1 -12546.196,E2 -12546.196} C_VEL
LIN {X 0,Y 368.902,Z 216.157,A -85,B 0,C 180,E1 -12548.952,E2 -12548.952} C_VEL
LIN {X 0,Y 368.879,Z 216.16,A -85,B 0,C 180,E1 -12552.009,E2 -12552.009} C_VEL
LIN {X 0,Y 368.923,Z 216.157,A -85,B 0,C 180,E1 -12555.182,E2 -12555.182} C_VEL
LIN {X 0,Y 368.89,Z 216.149,A -85,B 0,C 180,E1 -12558.178,E2 -12558.178} C_VEL
LIN {X 0,Y 368.908,Z 216.147,A -85,B 0,C 180,E1 -12561.358,E2 -12561.358} C_VEL
LIN {X 0,Y 368.931,Z 216.156,A -85,B 0,C 180,E1 -12565.146,E2 -12565.146} C_VEL
LIN {X 0,Y 368.924,Z 216.134,A -85,B 0,C 180,E1 -12569.046,E2 -12569.046} C_VEL
LIN {X 0,Y 368.981,Z 216.148,A -85,B 0,C 180,E1 -12571.564,E2 -12571.564} C_VEL
LIN {X 0,Y 368.951,Z 216.154,A -85,B 0,C 180,E1 -12575.224,E2 -12575.224} C_VEL
LIN {X 0,Y 368.931,Z 216.155,A -85,B 0,C 180,E1 -12578.973,E2 -12578.973} C_VEL
LIN {X 0,Y 368.983,Z 216.141,A -85,B 0,C 180,E1 -12582.257,E2 -12582.257} C_VEL
LIN {X 0,Y 369.03,Z 216.133,A -85,B 0,C 180,E1 -12586.227,E2 -12586.227} C_VEL
LIN {X 0,Y 369.06,Z 216.13,A -85,B 0,C 180,E1 -12590.131,E2 -12590.131} C_VEL
LIN {X 0,Y 369.155,Z 216.126,A -85,B 0,C 180,E1 -12592.341,E2 -12592.341} C_VEL
LIN {X 0,Y 369.135,Z 216.123,A -85,B 0,C 180,E1 -12594.537,E2 -12594.537} C_VEL
LIN {X 0,Y 369.311,Z 216.105,A -85,B 0,C 180,E1 -12597.819,E2 -12597.819} C_VEL
LIN {X 0,Y 369.452,Z 216.08,A -85,B 0,C 180,E1 -12600,E2 -12600} C_VEL
LIN {X 0,Y 369.311,Z 216.107,A -85,B 0,C 180,E1 -12602.181,E2 -12602.181} C_VEL
LIN {X 0,Y 369.193,Z 216.125,A -85,B 0,C 180,E1 -12606.558,E2 -12606.558} C_VEL
LIN {X 0,Y 369.06,Z 216.135,A -85,B 0,C 180,E1 -12609.868,E2 -12609.868} C_VEL
LIN {X 0,Y 369.029,Z 216.137,A -85,B 0,C 180,E1 -12613.772,E2 -12613.772} C_VEL
LIN {X 0,Y 368.971,Z 216.145,A -85,B 0,C 180,E1 -12616.601,E2 -12616.601} C_VEL
LIN {X 0,Y 368.93,Z 216.158,A -85,B 0,C 180,E1 -12620.053,E2 -12620.053} C_VEL
LIN {X 0,Y 368.938,Z 216.156,A -85,B 0,C 180,E1 -12623.887,E2 -12623.887} C_VEL
LIN {X 0,Y 368.964,Z 216.15,A -85,B 0,C 180,E1 -12627.203,E2 -12627.203} C_VEL
LIN {X 0,Y 368.917,Z 216.157,A -85,B 0,C 180,E1 -12629.69,E2 -12629.69} C_VEL
LIN {X 0,Y 368.893,Z 216.153,A -85,B 0,C 180,E1 -12633.538,E2 -12633.538} C_VEL
LIN {X 0,Y 368.895,Z 216.157,A -85,B 0,C 180,E1 -12636.856,E2 -12636.856} C_VEL
LIN {X 0,Y 368.905,Z 216.137,A -85,B 0,C 180,E1 -12640.371,E2 -12640.371} C_VEL
LIN {X 0,Y 368.877,Z 216.162,A -85,B 0,C 180,E1 -12643.616,E2 -12643.616} C_VEL
LIN {X 0,Y 368.898,Z 216.157,A -85,B 0,C 180,E1 -12646.699,E2 -12646.699} C_VEL
LIN {X 0,Y 368.949,Z 216.151,A -85,B 0,C 180,E1 -12649.636,E2 -12649.636} C_VEL
LIN {X 0,Y 368.928,Z 216.214,A -85,B 0,C 180,E1 -12653.485,E2 -12653.485} C_VEL
LIN {X 0,Y 372.025,Z 227.601,A -85,B 0,C 180,E1 -12656.223,E2 -12656.223} C_VEL
LIN {X 0,Y 375.197,Z 240.368,A -85,B 0,C 180,E1 -12659.105,E2 -12659.105} C_VEL
LIN {X 0,Y 380.834,Z 253.478,A -85,B 0,C 180,E1 -12659.887,E2 -12659.887} C_VEL
LIN {X 0,Y 386.075,Z 280.609,A -85,B 0,C 180,E1 -12660.9,E2 -12660.9} C_VEL
LIN {X 0,Y 386.256,Z 285.256,A -85,B 0,C 180,E1 -12661.012,E2 -12661.012} C_VEL
LIN {X 0,Y 383.274,Z 406.279,A -85,B 0,C 180,E1 -12663.305,E2 -12663.305} C_VEL
LIN {X 0,Y 382.465,Z 421.759,A -85,B 0,C 180,E1 -12663.795,E2 -12663.795} C_VEL
LIN {X 0,Y 381.31,Z 435.402,A -85,B 0,C 180,E1 -12664.408,E2 -12664.408} C_VEL
LIN {X 0,Y 380.026,Z 448.794,A -85,B 0,C 180,E1 -12665.2,E2 -12665.2} C_VEL
LIN {X 0,Y 378.454,Z 461.998,A -85,B 0,C 180,E1 -12666.178,E2 -12666.178} C_VEL
LIN {X 0,Y 376.754,Z 475.022,A -85,B 0,C 180,E1 -12667.373,E2 -12667.373} C_VEL
LIN {X 0,Y 375.098,Z 487.054,A -85,B 0,C 180,E1 -12668.715,E2 -12668.715} C_VEL
LIN {X 0,Y 373.475,Z 498.202,A -85,B 0,C 180,E1 -12670.202,E2 -12670.202} C_VEL
LIN {X 0,Y 372.023,Z 508.466,A -85,B 0,C 180,E1 -12671.838,E2 -12671.838} C_VEL
LIN {X 0,Y 370.522,Z 518.498,A -85,B 0,C 180,E1 -12673.754,E2 -12673.754} C_VEL
LIN {X 0,Y 369.357,Z 526.835,A -85,B 0,C 180,E1 -12675.679,E2 -12675.679} C_VEL
LIN {X 0,Y 368.549,Z 534.675,A -85,B 0,C 180,E1 -12677.892,E2 -12677.892} C_VEL
LIN {X 0,Y 367.867,Z 540.912,A -85,B 0,C 180,E1 -12680.099,E2 -12680.099} C_VEL
LIN {X 0,Y 367.573,Z 545.741,A -85,B 0,C 180,E1 -12682.309,E2 -12682.309} C_VEL
LIN {X 0,Y 367.41,Z 549.28,A -85,B 0,C 180,E1 -12684.512,E2 -12684.512} C_VEL
LIN {X 0,Y 367.352,Z 551.609,A -85,B 0,C 180,E1 -12686.71,E2 -12686.71} C_VEL
LIN {X 0,Y 367.414,Z 552.781,A -85,B 0,C 180,E1 -12688.904,E2 -12688.904} C_VEL
LIN {X 0,Y 367.414,Z 552.779,A -85,B 0,C 180,E1 -12691.096,E2 -12691.096} C_VEL
LIN {X 0,Y 367.352,Z 551.597,A -85,B 0,C 180,E1 -12693.29,E2 -12693.29} C_VEL
LIN {X 0,Y 367.41,Z 549.262,A -85,B 0,C 180,E1 -12695.488,E2 -12695.488} C_VEL
LIN {X 0,Y 367.573,Z 545.723,A -85,B 0,C 180,E1 -12697.691,E2 -12697.691} C_VEL
LIN {X 0,Y 367.867,Z 540.889,A -85,B 0,C 180,E1 -12699.901,E2 -12699.901} C_VEL
LIN {X 0,Y 368.542,Z 534.637,A -85,B 0,C 180,E1 -12702.108,E2 -12702.108} C_VEL
LIN {X 0,Y 369.356,Z 526.785,A -85,B 0,C 180,E1 -12704.321,E2 -12704.321} C_VEL
LIN {X 0,Y 370.523,Z 518.443,A -85,B 0,C 180,E1 -12706.246,E2 -12706.246} C_VEL
LIN {X 0,Y 372.038,Z 508.399,A -85,B 0,C 180,E1 -12708.161,E2 -12708.161} C_VEL
LIN {X 0,Y 373.475,Z 498.128,A -85,B 0,C 180,E1 -12709.798,E2 -12709.798} C_VEL
LIN {X 0,Y 375.233,Z 485.894,A -85,B 0,C 180,E1 -12711.421,E2 -12711.421} C_VEL
LIN {X 0,Y 377.122,Z 472.279,A -85,B 0,C 180,E1 -12712.893,E2 -12712.893} C_VEL
LIN {X 0,Y 378.856,Z 458.63,A -85,B 0,C 180,E1 -12714.086,E2 -12714.086} C_VEL
LIN {X 0,Y 380.376,Z 445.144,A -85,B 0,C 180,E1 -12715.029,E2 -12715.029} C_VEL
LIN {X 0,Y 381.687,Z 430.61,A -85,B 0,C 180,E1 -12715.822,E2 -12715.822} C_VEL
LIN {X 0,Y 382.786,Z 415.017,A -85,B 0,C 180,E1 -12716.438,E2 -12716.438} C_VEL
LIN {X 0,Y 383.5,Z 399.698,A -85,B 0,C 180,E1 -12716.825,E2 -12716.825} C_VEL
LIN {X 0,Y 386.299,Z 282.501,A -85,B 0,C 180,E1 -12719.027,E2 -12719.027} C_VEL
LIN {X 0,Y 381.247,Z 255.319,A -85,B 0,C 180,E1 -12720.022,E2 -12720.022} C_VEL
LIN {X 0,Y 379.984,Z 251.104,A -85,B 0,C 180,E1 -12720.221,E2 -12720.221} C_VEL
LIN {X 0,Y 375.151,Z 240.158,A -85,B 0,C 180,E1 -12720.901,E2 -12720.901} C_VEL
LIN {X 0,Y 371.693,Z 226.351,A -85,B 0,C 180,E1 -12724.05,E2 -12724.05} C_VEL
LIN {X 0,Y 368.928,Z 216.152,A -85,B 0,C 180,E1 -12726.515,E2 -12726.515} C_VEL
LIN {X 0,Y 368.949,Z 216.154,A -85,B 0,C 180,E1 -12730.364,E2 -12730.364} C_VEL
LIN {X 0,Y 368.89,Z 216.158,A -85,B 0,C 180,E1 -12733.617,E2 -12733.617} C_VEL
LIN {X 0,Y 368.898,Z 216.154,A -85,B 0,C 180,E1 -12736.698,E2 -12736.698} C_VEL
LIN {X 0,Y 368.948,Z 216.147,A -85,B 0,C 180,E1 -12739.635,E2 -12739.635} C_VEL
LIN {X 0,Y 368.897,Z 216.153,A -85,B 0,C 180,E1 -12743.143,E2 -12743.143} C_VEL
LIN {X 0,Y 368.895,Z 216.151,A -85,B 0,C 180,E1 -12746.462,E2 -12746.462} C_VEL
LIN {X 0,Y 368.917,Z 216.151,A -85,B 0,C 180,E1 -12750.31,E2 -12750.31} C_VEL
LIN {X 0,Y 368.975,Z 216.145,A -85,B 0,C 180,E1 -12753.535,E2 -12753.535} C_VEL
LIN {X 0,Y 368.949,Z 216.144,A -85,B 0,C 180,E1 -12756.421,E2 -12756.421} C_VEL
LIN {X 0,Y 368.923,Z 216.145,A -85,B 0,C 180,E1 -12759.946,E2 -12759.946} C_VEL
LIN {X 0,Y 368.968,Z 216.146,A -85,B 0,C 180,E1 -12763.398,E2 -12763.398} C_VEL
LIN {X 0,Y 369.05,Z 216.136,A -85,B 0,C 180,E1 -12766.79,E2 -12766.79} C_VEL
LIN {X 0,Y 369.06,Z 216.136,A -85,B 0,C 180,E1 -12770.132,E2 -12770.132} C_VEL
LIN {X 0,Y 369.193,Z 216.124,A -85,B 0,C 180,E1 -12773.442,E2 -12773.442} C_VEL
LIN {X 0,Y 369.311,Z 216.107,A -85,B 0,C 180,E1 -12777.819,E2 -12777.819} C_VEL
LIN {X 0,Y 369.452,Z 216.082,A -85,B 0,C 180,E1 -12780,E2 -12780} C_VEL
LIN {X 0,Y 369.311,Z 216.105,A -85,B 0,C 180,E1 -12782.181,E2 -12782.181} C_VEL
LIN {X 0,Y 369.19,Z 216.12,A -85,B 0,C 180,E1 -12786.616,E2 -12786.616} C_VEL
LIN {X 0,Y 369.06,Z 216.137,A -85,B 0,C 180,E1 -12789.869,E2 -12789.869} C_VEL
LIN {X 0,Y 369.03,Z 216.141,A -85,B 0,C 180,E1 -12793.773,E2 -12793.773} C_VEL
LIN {X 0,Y 368.994,Z 216.145,A -85,B 0,C 180,E1 -12797.769,E2 -12797.769} C_VEL
LIN {X 0,Y 368.903,Z 216.155,A -85,B 0,C 180,E1 -12801.221,E2 -12801.221} C_VEL
LIN {X 0,Y 368.949,Z 216.137,A -85,B 0,C 180,E1 -12804.776,E2 -12804.776} C_VEL
LIN {X 0,Y 368.965,Z 216.133,A -85,B 0,C 180,E1 -12807.203,E2 -12807.203} C_VEL
LIN {X 0,Y 368.917,Z 216.154,A -85,B 0,C 180,E1 -12809.69,E2 -12809.69} C_VEL
LIN {X 0,Y 368.891,Z 216.154,A -85,B 0,C 180,E1 -12813.539,E2 -12813.539} C_VEL
LIN {X 0,Y 368.897,Z 216.155,A -85,B 0,C 180,E1 -12816.857,E2 -12816.857} C_VEL
LIN {X 0,Y 368.906,Z 216.153,A -85,B 0,C 180,E1 -12820.371,E2 -12820.371} C_VEL
LIN {X 0,Y 368.88,Z 216.157,A -85,B 0,C 180,E1 -12823.617,E2 -12823.617} C_VEL
LIN {X 0,Y 368.883,Z 216.159,A -85,B 0,C 180,E1 -12826.697,E2 -12826.697} C_VEL
LIN {X 0,Y 368.909,Z 216.158,A -85,B 0,C 180,E1 -12829.644,E2 -12829.644} C_VEL
LIN {X 0,Y 368.899,Z 216.158,A -85,B 0,C 180,E1 -12833.145,E2 -12833.145} C_VEL
LIN {X 0,Y 368.895,Z 216.154,A -85,B 0,C 180,E1 -12836.463,E2 -12836.463} C_VEL
LIN {X 0,Y 368.898,Z 216.16,A -85,B 0,C 180,E1 -12837.054,E2 -12837.054} C_VEL
LIN {X 0,Y 370.62,Z 222.677,A -85,B 0,C 180,E1 -12838.749,E2 -12838.749} C_VEL
LIN {X 0,Y 381.87,Z 245.967,A -85,B 0,C 180,E1 -12840.276,E2 -12840.276} C_VEL
LIN {X 0,Y 386.677,Z 257.465,A -85,B 0,C 180,E1 -12840.925,E2 -12840.925} C_VEL
LIN {X 0,Y 384.557,Z 353.287,A -85,B 0,C 180,E1 -12842.742,E2 -12842.742} C_VEL
LIN {X 0,Y 383.561,Z 388.617,A -85,B 0,C 180,E1 -12843.437,E2 -12843.437} C_VEL
LIN {X 0,Y 382.787,Z 403.547,A -85,B 0,C 180,E1 -12843.932,E2 -12843.932} C_VEL
LIN {X 0,Y 381.79,Z 417.517,A -85,B 0,C 180,E1 -12844.59,E2 -12844.59} C_VEL
LIN {X 0,Y 380.547,Z 431.323,A -85,B 0,C 180,E1 -12845.448,E2 -12845.448} C_VEL
LIN {X 0,Y 379.038,Z 444.896,A -85,B 0,C 180,E1 -12846.507,E2 -12846.507} C_VEL
LIN {X 0,Y 377.408,Z 457.379,A -85,B 0,C 180,E1 -12847.703,E2 -12847.703} C_VEL
LIN {X 0,Y 375.636,Z 470.02,A -85,B 0,C 180,E1 -12849.178,E2 -12849.178} C_VEL
LIN {X 0,Y 373.956,Z 481.478,A -85,B 0,C 180,E1 -12850.799,E2 -12850.799} C_VEL
LIN {X 0,Y 372.497,Z 491.116,A -85,B 0,C 180,E1 -12852.43,E2 -12852.43} C_VEL
LIN {X 0,Y 371.079,Z 500.561,A -85,B 0,C 180,E1 -12854.343,E2 -12854.343} C_VEL
LIN {X 0,Y 369.966,Z 508.42,A -85,B 0,C 180,E1 -12856.264,E2 -12856.264} C_VEL
LIN {X 0,Y 369.171,Z 514.084,A -85,B 0,C 180,E1 -12857.913,E2 -12857.913} C_VEL
LIN {X 0,Y 368.417,Z 520.253,A -85,B 0,C 180,E1 -12860.114,E2 -12860.114} C_VEL
LIN {X 0,Y 367.956,Z 525.014,A -85,B 0,C 180,E1 -12862.317,E2 -12862.317} C_VEL
LIN {X 0,Y 367.673,Z 528.502,A -85,B 0,C 180,E1 -12864.516,E2 -12864.516} C_VEL
LIN {X 0,Y 367.452,Z 530.81,A -85,B 0,C 180,E1 -12866.711,E2 -12866.711} C_VEL
LIN {X 0,Y 367.445,Z 531.986,A -85,B 0,C 180,E1 -12868.904,E2 -12868.904} C_VEL
LIN {X 0,Y 367.445,Z 532.001,A -85,B 0,C 180,E1 -12871.096,E2 -12871.096} C_VEL
LIN {X 0,Y 367.451,Z 530.886,A -85,B 0,C 180,E1 -12873.289,E2 -12873.289} C_VEL
LIN {X 0,Y 367.66,Z 528.638,A -85,B 0,C 180,E1 -12875.484,E2 -12875.484} C_VEL
LIN {X 0,Y 367.952,Z 524.793,A -85,B 0,C 180,E1 -12877.9,E2 -12877.9} C_VEL
LIN {X 0,Y 368.408,Z 520.506,A -85,B 0,C 180,E1 -12879.886,E2 -12879.886} C_VEL
LIN {X 0,Y 369.16,Z 514.413,A -85,B 0,C 180,E1 -12882.088,E2 -12882.088} C_VEL
LIN {X 0,Y 369.29,Z 513.639,A -85,B 0,C 180,E1 -12882.324,E2 -12882.324} C_VEL
LIN {X 0,Y 369.059,Z 511.038,A -85,B 0,C 180,E1 -12883.144,E2 -12883.144} C_VEL
LIN {X 0,Y 366.858,Z 506.645,A -85,B 0,C 180,E1 -12884.491,E2 -12884.491} C_VEL
LIN {X 0,Y 364.723,Z 501.837,A -85,B 0,C 180,E1 -12885.811,E2 -12885.811} C_VEL
LIN {X 0,Y 364.592,Z 498.483,A -85,B 0,C 180,E1 -12886.576,E2 -12886.576} C_VEL
LIN {X 0,Y 366.135,Z 488.886,A -85,B 0,C 180,E1 -12888.464,E2 -12888.464} C_VEL
LIN {X 0,Y 367.952,Z 477.359,A -85,B 0,C 180,E1 -12890.331,E2 -12890.331} C_VEL
LIN {X 0,Y 369.714,Z 465.613,A -85,B 0,C 180,E1 -12891.904,E2 -12891.904} C_VEL
LIN {X 0,Y 371.464,Z 453.336,A -85,B 0,C 180,E1 -12893.262,E2 -12893.262} C_VEL
LIN {X 0,Y 373.178,Z 439.912,A -85,B 0,C 180,E1 -12894.476,E2 -12894.476} C_VEL
LIN {X 0,Y 374.749,Z 424.949,A -85,B 0,C 180,E1 -12895.552,E2 -12895.552} C_VEL
LIN {X 0,Y 376.027,Z 409.633,A -85,B 0,C 180,E1 -12896.389,E2 -12896.389} C_VEL
LIN {X 0,Y 377.035,Z 394.294,A -85,B 0,C 180,E1 -12896.985,E2 -12896.985} C_VEL
LIN {X 0,Y 377.641,Z 378.077,A -85,B 0,C 180,E1 -12897.388,E2 -12897.388} C_VEL
LIN {X 0,Y 380.082,Z 279.397,A -85,B 0,C 180,E1 -12899.273,E2 -12899.273} C_VEL
LIN {X 0,Y 380.45,Z 259.386,A -85,B 0,C 180,E1 -12899.667,E2 -12899.667} C_VEL
LIN {X 0,Y 374.441,Z 245.497,A -85,B 0,C 180,E1 -12900.499,E2 -12900.499} C_VEL
LIN {X 0,Y 365.238,Z 226.531,A -85,B 0,C 180,E1 -12901.789,E2 -12901.789} C_VEL
LIN {X 0,Y 363.382,Z 222.866,A -85,B 0,C 180,E1 -12902.065,E2 -12902.065} C_VEL
LIN {X 0,Y 361.871,Z 217.034,A -85,B 0,C 180,E1 -12903.646,E2 -12903.646} C_VEL
LIN {X 0,Y 361.863,Z 217.033,A -85,B 0,C 180,E1 -12907.222,E2 -12907.222} C_VEL
LIN {X 0,Y 361.833,Z 217.036,A -85,B 0,C 180,E1 -12910.755,E2 -12910.755} C_VEL
LIN {X 0,Y 361.818,Z 217.038,A -85,B 0,C 180,E1 -12914.367,E2 -12914.367} C_VEL
LIN {X 0,Y 361.838,Z 217.025,A -85,B 0,C 180,E1 -12917.566,E2 -12917.566} C_VEL
LIN {X 0,Y 361.87,Z 217.029,A -85,B 0,C 180,E1 -12920.972,E2 -12920.972} C_VEL
LIN {X 0,Y 361.869,Z 217.03,A -85,B 0,C 180,E1 -12924.654,E2 -12924.654} C_VEL
LIN {X 0,Y 361.832,Z 217.015,A -85,B 0,C 180,E1 -12928.37,E2 -12928.37} C_VEL
LIN {X 0,Y 361.896,Z 217.027,A -85,B 0,C 180,E1 -12930.955,E2 -12930.955} C_VEL
LIN {X 0,Y 361.948,Z 217.018,A -85,B 0,C 180,E1 -12933.474,E2 -12933.474} C_VEL
LIN {X 0,Y 361.883,Z 217.027,A -85,B 0,C 180,E1 -12937.144,E2 -12937.144} C_VEL
LIN {X 0,Y 361.899,Z 217.027,A -85,B 0,C 180,E1 -12940.723,E2 -12940.723} C_VEL
LIN {X 0,Y 361.926,Z 217.029,A -85,B 0,C 180,E1 -12943.066,E2 -12943.066} C_VEL
